LIN {X 0,Y 256.151,Z 298.388,A -85,B 0,C 180,E1 -18561.12,E2 -18561.12} C_VEL
LIN {X 0,Y 256.183,Z 298.389,A -85,B 0,C 180,E1 -18565.139,E2 -18565.139} C_VEL
LIN {X 0,Y 256.099,Z 298.396,A -85,B 0,C 180,E1 -18569.602,E2 -18569.602} C_VEL
LIN {X 0,Y 256.137,Z 298.525,A -85,B 0,C 180,E1 -18573.387,E2 -18573.387} C_VEL
LIN {X 0,Y 256.985,Z 302.055,A -85,B 0,C 180,E1 -18575.051,E2 -18575.051} C_VEL
LIN {X 0,Y 263.939,Z 316.937,A -85,B 0,C 180,E1 -18576.488,E2 -18576.488} C_VEL
LIN {X 0,Y 267.967,Z 326.974,A -85,B 0,C 180,E1 -18577.308,E2 -18577.308} C_VEL
LIN {X 0,Y 269.292,Z 334.674,A -85,B 0,C 180,E1 -18577.711,E2 -18577.711} C_VEL
LIN {X 0,Y 267.661,Z 378.993,A -85,B 0,C 180,E1 -18578.986,E2 -18578.986} C_VEL
LIN {X 0,Y 266.948,Z 389.558,A -85,B 0,C 180,E1 -18579.509,E2 -18579.509} C_VEL
LIN {X 0,Y 265.887,Z 401.083,A -85,B 0,C 180,E1 -18580.395,E2 -18580.395} C_VEL
LIN {X 0,Y 264.658,Z 410.377,A -85,B 0,C 180,E1 -18581.383,E2 -18581.383} C_VEL
LIN {X 0,Y 263.326,Z 418.675,A -85,B 0,C 180,E1 -18582.501,E2 -18582.501} C_VEL
LIN {X 0,Y 262.135,Z 425.481,A -85,B 0,C 180,E1 -18583.626,E2 -18583.626} C_VEL
LIN {X 0,Y 260.662,Z 432.609,A -85,B 0,C 180,E1 -18585.053,E2 -18585.053} C_VEL
LIN {X 0,Y 259.485,Z 437.896,A -85,B 0,C 180,E1 -18586.321,E2 -18586.321} C_VEL
LIN {X 0,Y 258.097,Z 444.114,A -85,B 0,C 180,E1 -18588.155,E2 -18588.155} C_VEL
LIN {X 0,Y 257.179,Z 448.17,A -85,B 0,C 180,E1 -18589.609,E2 -18589.609} C_VEL
LIN {X 0,Y 256.425,Z 451.313,A -85,B 0,C 180,E1 -18590.924,E2 -18590.924} C_VEL
LIN {X 0,Y 255.519,Z 455.024,A -85,B 0,C 180,E1 -18592.906,E2 -18592.906} C_VEL
LIN {X 0,Y 254.875,Z 457.473,A -85,B 0,C 180,E1 -18594.617,E2 -18594.617} C_VEL
LIN {X 0,Y 254.468,Z 459.361,A -85,B 0,C 180,E1 -18596.472,E2 -18596.472} C_VEL
LIN {X 0,Y 253.925,Z 460.797,A -85,B 0,C 180,E1 -18599.093,E2 -18599.093} C_VEL
LIN {X 0,Y 253.67,Z 460.823,A -85,B 0,C 180,E1 -18601.902,E2 -18601.902} C_VEL
LIN {X 0,Y 253.733,Z 460.029,A -85,B 0,C 180,E1 -18603.694,E2 -18603.694} C_VEL
LIN {X 0,Y 254.011,Z 458.128,A -85,B 0,C 180,E1 -18605.93,E2 -18605.93} C_VEL
LIN {X 0,Y 254.428,Z 455.249,A -85,B 0,C 180,E1 -18608.106,E2 -18608.106} C_VEL
LIN {X 0,Y 255.092,Z 450.342,A -85,B 0,C 180,E1 -18610.695,E2 -18610.695} C_VEL
LIN {X 0,Y 255.797,Z 444.962,A -85,B 0,C 180,E1 -18612.77,E2 -18612.77} C_VEL
LIN {X 0,Y 256.639,Z 439.307,A -85,B 0,C 180,E1 -18614.515,E2 -18614.515} C_VEL
LIN {X 0,Y 257.604,Z 432.621,A -85,B 0,C 180,E1 -18616.19,E2 -18616.19} C_VEL
LIN {X 0,Y 258.639,Z 425.015,A -85,B 0,C 180,E1 -18617.738,E2 -18617.738} C_VEL
LIN {X 0,Y 259.909,Z 415.481,A -85,B 0,C 180,E1 -18619.287,E2 -18619.287} C_VEL
LIN {X 0,Y 260.987,Z 405.524,A -85,B 0,C 180,E1 -18620.507,E2 -18620.507} C_VEL
LIN {X 0,Y 261.726,Z 395.897,A -85,B 0,C 180,E1 -18621.411,E2 -18621.411} C_VEL
LIN {X 0,Y 262.374,Z 386.398,A -85,B 0,C 180,E1 -18622.062,E2 -18622.062} C_VEL
LIN {X 0,Y 262.898,Z 376.662,A -85,B 0,C 180,E1 -18622.506,E2 -18622.506} C_VEL
LIN {X 0,Y 263.995,Z 331.197,A -85,B 0,C 180,E1 -18623.814,E2 -18623.814} C_VEL
LIN {X 0,Y 260.762,Z 313.544,A -85,B 0,C 180,E1 -18624.586,E2 -18624.586} C_VEL
LIN {X 0,Y 257.013,Z 301.84,A -85,B 0,C 180,E1 -18625.25,E2 -18625.25} C_VEL
LIN {X 0,Y 256.516,Z 298.349,A -85,B 0,C 180,E1 -18626.859,E2 -18626.859} C_VEL
LIN {X 0,Y 256.767,Z 298.316,A -85,B 0,C 180,E1 -18630,E2 -18630} C_VEL
LIN {X 0,Y 256.498,Z 298.345,A -85,B 0,C 180,E1 -18633.141,E2 -18633.141} C_VEL
LIN {X 0,Y 256.498,Z 298.346,A -85,B 0,C 180,E1 -18637.874,E2 -18637.874} C_VEL
LIN {X 0,Y 256.291,Z 298.369,A -85,B 0,C 180,E1 -18642.672,E2 -18642.672} C_VEL
LIN {X 0,Y 256.244,Z 298.379,A -85,B 0,C 180,E1 -18646.271,E2 -18646.271} C_VEL
LIN {X 0,Y 256.142,Z 298.377,A -85,B 0,C 180,E1 -18651.11,E2 -18651.11} C_VEL
LIN {X 0,Y 256.17,Z 298.388,A -85,B 0,C 180,E1 -18655.129,E2 -18655.129} C_VEL
LIN {X 0,Y 256.113,Z 298.394,A -85,B 0,C 180,E1 -18659.599,E2 -18659.599} C_VEL
LIN {X 0,Y 256.067,Z 298.399,A -85,B 0,C 180,E1 -18663.292,E2 -18663.292} C_VEL
LIN {X 0,Y 256.112,Z 298.398,A -85,B 0,C 180,E1 -18667.27,E2 -18667.27} C_VEL
LIN {X 0,Y 256.057,Z 298.4,A -85,B 0,C 180,E1 -18671.201,E2 -18671.201} C_VEL
LIN {X 0,Y 256.073,Z 298.399,A -85,B 0,C 180,E1 -18675.525,E2 -18675.525} C_VEL
LIN {X 0,Y 256.1,Z 298.394,A -85,B 0,C 180,E1 -18678.805,E2 -18678.805} C_VEL
LIN {X 0,Y 256.149,Z 298.383,A -85,B 0,C 180,E1 -18682.87,E2 -18682.87} C_VEL
LIN {X 0,Y 256.08,Z 298.391,A -85,B 0,C 180,E1 -18686.709,E2 -18686.709} C_VEL
LIN {X 0,Y 256.13,Z 298.39,A -85,B 0,C 180,E1 -18691.405,E2 -18691.405} C_VEL
LIN {X 0,Y 256.161,Z 298.384,A -85,B 0,C 180,E1 -18695.698,E2 -18695.698} C_VEL
LIN {X 0,Y 256.16,Z 298.374,A -85,B 0,C 180,E1 -18699.104,E2 -18699.104} C_VEL
LIN {X 0,Y 256.287,Z 298.369,A -85,B 0,C 180,E1 -18704.084,E2 -18704.084} C_VEL
LIN {X 0,Y 256.286,Z 298.371,A -85,B 0,C 180,E1 -18707.327,E2 -18707.327} C_VEL
LIN {X 0,Y 256.507,Z 298.339,A -85,B 0,C 180,E1 -18712.126,E2 -18712.126} C_VEL
LIN {X 0,Y 256.488,Z 298.34,A -85,B 0,C 180,E1 -18716.858,E2 -18716.858} C_VEL
LIN {X 0,Y 256.757,Z 298.31,A -85,B 0,C 180,E1 -18720,E2 -18720} C_VEL
LIN {X 0,Y 256.488,Z 298.35,A -85,B 0,C 180,E1 -18723.141,E2 -18723.141} C_VEL
LIN {X 0,Y 256.507,Z 298.337,A -85,B 0,C 180,E1 -18727.874,E2 -18727.874} C_VEL
LIN {X 0,Y 256.287,Z 298.368,A -85,B 0,C 180,E1 -18732.672,E2 -18732.672} C_VEL
LIN {X 0,Y 256.27,Z 298.375,A -85,B 0,C 180,E1 -18735.88,E2 -18735.88} C_VEL
LIN {X 0,Y 255.651,Z 298.459,A -85,B 0,C 180,E1 -18737.191,E2 -18737.191} C_VEL
LIN {X 0,Y 252.715,Z 298.819,A -85,B 0,C 180,E1 -18739.322,E2 -18739.322} C_VEL
LIN {X 0,Y 250.187,Z 299.124,A -85,B 0,C 180,E1 -18741.059,E2 -18741.059} C_VEL
LIN {X 0,Y 249.116,Z 299.262,A -85,B 0,C 180,E1 -18742.409,E2 -18742.409} C_VEL
LIN {X 0,Y 249.039,Z 299.268,A -85,B 0,C 180,E1 -18742.867,E2 -18742.867} C_VEL
LIN {X 0,Y 249.11,Z 299.265,A -85,B 0,C 180,E1 -18745.476,E2 -18745.476} C_VEL
LIN {X 0,Y 249.067,Z 299.268,A -85,B 0,C 180,E1 -18748.989,E2 -18748.989} C_VEL
LIN {X 0,Y 249.025,Z 299.279,A -85,B 0,C 180,E1 -18752.426,E2 -18752.426} C_VEL
LIN {X 0,Y 249.042,Z 299.277,A -85,B 0,C 180,E1 -18756.343,E2 -18756.343} C_VEL
LIN {X 0,Y 249.001,Z 299.27,A -85,B 0,C 180,E1 -18760.479,E2 -18760.479} C_VEL
LIN {X 0,Y 249.003,Z 299.282,A -85,B 0,C 180,E1 -18764.879,E2 -18764.879} C_VEL
LIN {X 0,Y 249.014,Z 299.277,A -85,B 0,C 180,E1 -18767.364,E2 -18767.364} C_VEL
LIN {X 0,Y 249.04,Z 299.274,A -85,B 0,C 180,E1 -18772.201,E2 -18772.201} C_VEL
LIN {X 0,Y 249.04,Z 299.274,A -85,B 0,C 180,E1 -18775.64,E2 -18775.64} C_VEL
LIN {X 0,Y 249.104,Z 299.285,A -85,B 0,C 180,E1 -18779.681,E2 -18779.681} C_VEL
LIN {X 0,Y 250.677,Z 307.76,A -85,B 0,C 180,E1 -18783.348,E2 -18783.348} C_VEL
LIN {X 0,Y 251.627,Z 313.3,A -85,B 0,C 180,E1 -18785.672,E2 -18785.672} C_VEL
LIN {X 0,Y 251.442,Z 315.01,A -85,B 0,C 180,E1 -18786.346,E2 -18786.346} C_VEL
LIN {X 0,Y 256.334,Z 351.638,A -85,B 0,C 180,E1 -18787.87,E2 -18787.87} C_VEL
LIN {X 0,Y 256.775,Z 358.082,A -85,B 0,C 180,E1 -18788.1,E2 -18788.1} C_VEL
LIN {X 0,Y 255.846,Z 392.247,A -85,B 0,C 180,E1 -18789.13,E2 -18789.13} C_VEL
LIN {X 0,Y 255.2,Z 402.545,A -85,B 0,C 180,E1 -18789.652,E2 -18789.652} C_VEL
LIN {X 0,Y 254.459,Z 410.782,A -85,B 0,C 180,E1 -18790.259,E2 -18790.259} C_VEL
LIN {X 0,Y 253.319,Z 422.12,A -85,B 0,C 180,E1 -18791.395,E2 -18791.395} C_VEL
LIN {X 0,Y 252.082,Z 432.063,A -85,B 0,C 180,E1 -18792.77,E2 -18792.77} C_VEL
LIN {X 0,Y 250.974,Z 440.032,A -85,B 0,C 180,E1 -18794.156,E2 -18794.156} C_VEL
LIN {X 0,Y 249.886,Z 447.476,A -85,B 0,C 180,E1 -18795.754,E2 -18795.754} C_VEL
LIN {X 0,Y 248.779,Z 455.022,A -85,B 0,C 180,E1 -18797.768,E2 -18797.768} C_VEL
LIN {X 0,Y 247.969,Z 460.929,A -85,B 0,C 180,E1 -18799.797,E2 -18799.797} C_VEL
LIN {X 0,Y 247.384,Z 465.565,A -85,B 0,C 180,E1 -18801.834,E2 -18801.834} C_VEL
LIN {X 0,Y 247.098,Z 468.571,A -85,B 0,C 180,E1 -18803.468,E2 -18803.468} C_VEL
LIN {X 0,Y 246.923,Z 470.901,A -85,B 0,C 180,E1 -18805.102,E2 -18805.102} C_VEL
LIN {X 0,Y 246.907,Z 472.628,A -85,B 0,C 180,E1 -18806.737,E2 -18806.737} C_VEL
LIN {X 0,Y 246.931,Z 473.843,A -85,B 0,C 180,E1 -18808.369,E2 -18808.369} C_VEL
LIN {X 0,Y 246.981,Z 474.572,A -85,B 0,C 180,E1 -18810,E2 -18810} C_VEL
LIN {X 0,Y 246.907,Z 474.817,A -85,B 0,C 180,E1 -18811.631,E2 -18811.631} C_VEL
LIN {X 0,Y 246.88,Z 474.471,A -85,B 0,C 180,E1 -18813.264,E2 -18813.264} C_VEL
LIN {X 0,Y 246.943,Z 473.512,A -85,B 0,C 180,E1 -18815.063,E2 -18815.063} C_VEL
LIN {X 0,Y 247.126,Z 472.282,A -85,B 0,C 180,E1 -18816.532,E2 -18816.532} C_VEL
LIN {X 0,Y 247.695,Z 469.279,A -85,B 0,C 180,E1 -18818.978,E2 -18818.978} C_VEL
LIN {X 0,Y 248.63,Z 465.018,A -85,B 0,C 180,E1 -18821.412,E2 -18821.412} C_VEL
LIN {X 0,Y 250.029,Z 459.189,A -85,B 0,C 180,E1 -18823.823,E2 -18823.823} C_VEL
LIN {X 0,Y 251.462,Z 452.925,A -85,B 0,C 180,E1 -18825.812,E2 -18825.812} C_VEL
LIN {X 0,Y 252.838,Z 446.82,A -85,B 0,C 180,E1 -18827.386,E2 -18827.386} C_VEL
LIN {X 0,Y 254.495,Z 439.407,A -85,B 0,C 180,E1 -18828.934,E2 -18828.934} C_VEL
LIN {X 0,Y 256.081,Z 431.486,A -85,B 0,C 180,E1 -18830.272,E2 -18830.272} C_VEL
LIN {X 0,Y 257.77,Z 421.644,A -85,B 0,C 180,E1 -18831.596,E2 -18831.596} C_VEL
LIN {X 0,Y 259.361,Z 410.129,A -85,B 0,C 180,E1 -18832.715,E2 -18832.715} C_VEL
LIN {X 0,Y 260.463,Z 400.369,A -85,B 0,C 180,E1 -18833.383,E2 -18833.383} C_VEL
LIN {X 0,Y 261.127,Z 391.422,A -85,B 0,C 180,E1 -18833.81,E2 -18833.81} C_VEL
LIN {X 0,Y 262.279,Z 357.245,A -85,B 0,C 180,E1 -18834.839,E2 -18834.839} C_VEL
LIN {X 0,Y 260.069,Z 341.118,A -85,B 0,C 180,E1 -18835.647,E2 -18835.647} C_VEL
LIN {X 0,Y 256.847,Z 324.506,A -85,B 0,C 180,E1 -18836.639,E2 -18836.639} C_VEL
LIN {X 0,Y 252.166,Z 313.492,A -85,B 0,C 180,E1 -18837.724,E2 -18837.724} C_VEL
LIN {X 0,Y 250.557,Z 305.695,A -85,B 0,C 180,E1 -18841.258,E2 -18841.258} C_VEL
LIN {X 0,Y 249.055,Z 299.276,A -85,B 0,C 180,E1 -18844.357,E2 -18844.357} C_VEL
LIN {X 0,Y 249.022,Z 299.285,A -85,B 0,C 180,E1 -18848.38,E2 -18848.38} C_VEL
LIN {X 0,Y 248.997,Z 299.285,A -85,B 0,C 180,E1 -18852.79,E2 -18852.79} C_VEL
LIN {X 0,Y 249.004,Z 299.283,A -85,B 0,C 180,E1 -18857.361,E2 -18857.361} C_VEL
LIN {X 0,Y 249.022,Z 299.274,A -85,B 0,C 180,E1 -18861.619,E2 -18861.619} C_VEL
LIN {X 0,Y 249.039,Z 299.275,A -85,B 0,C 180,E1 -18865.639,E2 -18865.639} C_VEL
LIN {X 0,Y 249.046,Z 299.273,A -85,B 0,C 180,E1 -18869.473,E2 -18869.473} C_VEL
LIN {X 0,Y 249.063,Z 299.258,A -85,B 0,C 180,E1 -18873.161,E2 -18873.161} C_VEL
LIN {X 0,Y 249.054,Z 299.267,A -85,B 0,C 180,E1 -18876.73,E2 -18876.73} C_VEL
LIN {X 0,Y 249.102,Z 299.263,A -85,B 0,C 180,E1 -18880.211,E2 -18880.211} C_VEL
LIN {X 0,Y 249.236,Z 299.237,A -85,B 0,C 180,E1 -18883.622,E2 -18883.622} C_VEL
LIN {X 0,Y 249.236,Z 299.246,A -85,B 0,C 180,E1 -18888.616,E2 -18888.616} C_VEL
LIN {X 0,Y 249.447,Z 299.214,A -85,B 0,C 180,E1 -18891.902,E2 -18891.902} C_VEL
LIN {X 0,Y 249.284,Z 299.235,A -85,B 0,C 180,E1 -18895.148,E2 -18895.148} C_VEL
LIN {X 0,Y 249.666,Z 299.189,A -85,B 0,C 180,E1 -18898.387,E2 -18898.387} C_VEL
LIN {X 0,Y 249.666,Z 299.183,A -85,B 0,C 180,E1 -18901.613,E2 -18901.613} C_VEL
LIN {X 0,Y 249.418,Z 299.222,A -85,B 0,C 180,E1 -18906.537,E2 -18906.537} C_VEL
LIN {X 0,Y 249.337,Z 299.24,A -85,B 0,C 180,E1 -18909.737,E2 -18909.737} C_VEL
LIN {X 0,Y 249.19,Z 299.258,A -85,B 0,C 180,E1 -18914.704,E2 -18914.704} C_VEL
LIN {X 0,Y 249.129,Z 299.266,A -85,B 0,C 180,E1 -18918.078,E2 -18918.078} C_VEL
LIN {X 0,Y 249.081,Z 299.271,A -85,B 0,C 180,E1 -18921.519,E2 -18921.519} C_VEL
LIN {X 0,Y 249.125,Z 299.27,A -85,B 0,C 180,E1 -18925.483,E2 -18925.483} C_VEL
LIN {X 0,Y 249.068,Z 299.27,A -85,B 0,C 180,E1 -18928.99,E2 -18928.99} C_VEL
LIN {X 0,Y 249.047,Z 299.309,A -85,B 0,C 180,E1 -18932.543,E2 -18932.543} C_VEL
LIN {X 0,Y 249.893,Z 302.544,A -85,B 0,C 180,E1 -18934.045,E2 -18934.045} C_VEL
LIN {X 0,Y 257.145,Z 317.447,A -85,B 0,C 180,E1 -18935.608,E2 -18935.608} C_VEL
LIN {X 0,Y 262.017,Z 329.387,A -85,B 0,C 180,E1 -18936.659,E2 -18936.659} C_VEL
LIN {X 0,Y 263.065,Z 335.339,A -85,B 0,C 180,E1 -18936.986,E2 -18936.986} C_VEL
LIN {X 0,Y 261.363,Z 379.31,A -85,B 0,C 180,E1 -18938.279,E2 -18938.279} C_VEL
LIN {X 0,Y 260.618,Z 390.029,A -85,B 0,C 180,E1 -18938.825,E2 -18938.825} C_VEL
LIN {X 0,Y 259.451,Z 401.845,A -85,B 0,C 180,E1 -18939.772,E2 -18939.772} C_VEL
LIN {X 0,Y 258.13,Z 411.2,A -85,B 0,C 180,E1 -18940.802,E2 -18940.802} C_VEL
LIN {X 0,Y 256.907,Z 418.493,A -85,B 0,C 180,E1 -18941.804,E2 -18941.804} C_VEL
LIN {X 0,Y 255.623,Z 425.55,A -85,B 0,C 180,E1 -18942.99,E2 -18942.99} C_VEL
LIN {X 0,Y 253.948,Z 433.158,A -85,B 0,C 180,E1 -18944.553,E2 -18944.553} C_VEL
LIN {X 0,Y 252.641,Z 438.698,A -85,B 0,C 180,E1 -18945.938,E2 -18945.938} C_VEL
LIN {X 0,Y 251.531,Z 443.472,A -85,B 0,C 180,E1 -18947.364,E2 -18947.364} C_VEL
LIN {X 0,Y 250.222,Z 448.785,A -85,B 0,C 180,E1 -18949.319,E2 -18949.319} C_VEL
LIN {X 0,Y 249.459,Z 451.837,A -85,B 0,C 180,E1 -18950.664,E2 -18950.664} C_VEL
LIN {X 0,Y 248.684,Z 454.871,A -85,B 0,C 180,E1 -18952.308,E2 -18952.308} C_VEL
LIN {X 0,Y 247.837,Z 457.857,A -85,B 0,C 180,E1 -18954.458,E2 -18954.458} C_VEL
LIN {X 0,Y 247.155,Z 460.258,A -85,B 0,C 180,E1 -18957.299,E2 -18957.299} C_VEL
LIN {X 0,Y 246.815,Z 461.045,A -85,B 0,C 180,E1 -18959.168,E2 -18959.168} C_VEL
LIN {X 0,Y 246.584,Z 460.961,A -85,B 0,C 180,E1 -18962.074,E2 -18962.074} C_VEL
LIN {X 0,Y 246.72,Z 459.547,A -85,B 0,C 180,E1 -18964.705,E2 -18964.705} C_VEL
LIN {X 0,Y 247.034,Z 457.72,A -85,B 0,C 180,E1 -18966.529,E2 -18966.529} C_VEL
LIN {X 0,Y 247.508,Z 454.157,A -85,B 0,C 180,E1 -18968.98,E2 -18968.98} C_VEL
LIN {X 0,Y 248.217,Z 449.125,A -85,B 0,C 180,E1 -18971.426,E2 -18971.426} C_VEL
LIN {X 0,Y 248.849,Z 444.55,A -85,B 0,C 180,E1 -18973.174,E2 -18973.174} C_VEL
LIN {X 0,Y 249.717,Z 438.959,A -85,B 0,C 180,E1 -18974.911,E2 -18974.911} C_VEL
LIN {X 0,Y 250.45,Z 434.013,A -85,B 0,C 180,E1 -18976.201,E2 -18976.201} C_VEL
LIN {X 0,Y 251.365,Z 427.852,A -85,B 0,C 180,E1 -18977.558,E2 -18977.558} C_VEL
LIN {X 0,Y 252.429,Z 420.063,A -85,B 0,C 180,E1 -18978.965,E2 -18978.965} C_VEL
LIN {X 0,Y 253.514,Z 411.395,A -85,B 0,C 180,E1 -18980.224,E2 -18980.224} C_VEL
LIN {X 0,Y 254.447,Z 402.338,A -85,B 0,C 180,E1 -18981.262,E2 -18981.262} C_VEL
LIN {X 0,Y 255.343,Z 390.86,A -85,B 0,C 180,E1 -18982.247,E2 -18982.247} C_VEL
LIN {X 0,Y 255.961,Z 380.029,A -85,B 0,C 180,E1 -18982.84,E2 -18982.84} C_VEL
LIN {X 0,Y 256.723,Z 354.048,A -85,B 0,C 180,E1 -18983.645,E2 -18983.645} C_VEL
LIN {X 0,Y 257.202,Z 331.869,A -85,B 0,C 180,E1 -18984.292,E2 -18984.292} C_VEL
LIN {X 0,Y 254.222,Z 315.471,A -85,B 0,C 180,E1 -18985.033,E2 -18985.033} C_VEL
LIN {X 0,Y 249.85,Z 301.947,A -85,B 0,C 180,E1 -18985.867,E2 -18985.867} C_VEL
LIN {X 0,Y 249.495,Z 299.225,A -85,B 0,C 180,E1 -18987.175,E2 -18987.175} C_VEL
LIN {X 0,Y 249.73,Z 299.193,A -85,B 0,C 180,E1 -18990,E2 -18990} C_VEL
LIN {X 0,Y 249.434,Z 299.225,A -85,B 0,C 180,E1 -18993.23,E2 -18993.23} C_VEL
LIN {X 0,Y 249.439,Z 299.225,A -85,B 0,C 180,E1 -18996.471,E2 -18996.471} C_VEL
LIN {X 0,Y 249.345,Z 299.238,A -85,B 0,C 180,E1 -18999.736,E2 -18999.736} C_VEL
LIN {X 0,Y 249.184,Z 299.258,A -85,B 0,C 180,E1 -19004.704,E2 -19004.704} C_VEL
LIN {X 0,Y 249.113,Z 299.265,A -85,B 0,C 180,E1 -19008.079,E2 -19008.079} C_VEL
LIN {X 0,Y 249.081,Z 299.254,A -85,B 0,C 180,E1 -19011.518,E2 -19011.518} C_VEL
LIN {X 0,Y 249.117,Z 299.265,A -85,B 0,C 180,E1 -19015.475,E2 -19015.475} C_VEL
LIN {X 0,Y 249.083,Z 299.274,A -85,B 0,C 180,E1 -19018.992,E2 -19018.992} C_VEL
LIN {X 0,Y 249.03,Z 299.273,A -85,B 0,C 180,E1 -19022.425,E2 -19022.425} C_VEL
LIN {X 0,Y 249.028,Z 299.276,A -85,B 0,C 180,E1 -19026.345,E2 -19026.345} C_VEL
LIN {X 0,Y 249.005,Z 299.276,A -85,B 0,C 180,E1 -19030.477,E2 -19030.477} C_VEL
LIN {X 0,Y 249.016,Z 299.274,A -85,B 0,C 180,E1 -19034.874,E2 -19034.874} C_VEL
LIN {X 0,Y 249.059,Z 299.273,A -85,B 0,C 180,E1 -19037.372,E2 -19037.372} C_VEL
LIN {X 0,Y 249.048,Z 299.273,A -85,B 0,C 180,E1 -19041.623,E2 -19041.623} C_VEL
LIN {X 0,Y 249.057,Z 299.263,A -85,B 0,C 180,E1 -19045.641,E2 -19045.641} C_VEL
LIN {X 0,Y 249.046,Z 299.272,A -85,B 0,C 180,E1 -19049.472,E2 -19049.472} C_VEL
LIN {X 0,Y 249.068,Z 299.269,A -85,B 0,C 180,E1 -19053.161,E2 -19053.161} C_VEL
LIN {X 0,Y 249.073,Z 299.263,A -85,B 0,C 180,E1 -19056.732,E2 -19056.732} C_VEL
LIN {X 0,Y 249.104,Z 299.255,A -85,B 0,C 180,E1 -19060.211,E2 -19060.211} C_VEL
LIN {X 0,Y 249.236,Z 299.246,A -85,B 0,C 180,E1 -19063.621,E2 -19063.621} C_VEL
LIN {X 0,Y 249.237,Z 299.253,A -85,B 0,C 180,E1 -19068.616,E2 -19068.616} C_VEL
LIN {X 0,Y 249.447,Z 299.218,A -85,B 0,C 180,E1 -19071.902,E2 -19071.902} C_VEL
LIN {X 0,Y 249.286,Z 299.234,A -85,B 0,C 180,E1 -19075.148,E2 -19075.148} C_VEL
LIN {X 0,Y 249.667,Z 299.191,A -85,B 0,C 180,E1 -19078.387,E2 -19078.387} C_VEL
LIN {X 0,Y 249.667,Z 299.196,A -85,B 0,C 180,E1 -19081.613,E2 -19081.613} C_VEL
LIN {X 0,Y 249.445,Z 299.219,A -85,B 0,C 180,E1 -19086.471,E2 -19086.471} C_VEL
LIN {X 0,Y 249.337,Z 299.231,A -85,B 0,C 180,E1 -19089.737,E2 -19089.737} C_VEL
LIN {X 0,Y 249.19,Z 299.254,A -85,B 0,C 180,E1 -19094.704,E2 -19094.704} C_VEL
LIN {X 0,Y 249.127,Z 299.262,A -85,B 0,C 180,E1 -19098.078,E2 -19098.078} C_VEL
LIN {X 0,Y 249.078,Z 299.264,A -85,B 0,C 180,E1 -19101.519,E2 -19101.519} C_VEL
LIN {X 0,Y 249.039,Z 299.268,A -85,B 0,C 180,E1 -19102.867,E2 -19102.867} C_VEL
LIN {X 0,Y 248.407,Z 299.355,A -85,B 0,C 180,E1 -19104.218,E2 -19104.218} C_VEL
LIN {X 0,Y 245.585,Z 299.71,A -85,B 0,C 180,E1 -19106.419,E2 -19106.419} C_VEL
LIN {X 0,Y 243.149,Z 300.01,A -85,B 0,C 180,E1 -19108.212,E2 -19108.212} C_VEL
LIN {X 0,Y 242.071,Z 300.14,A -85,B 0,C 180,E1 -19109.602,E2 -19109.602} C_VEL
LIN {X 0,Y 241.966,Z 300.15,A -85,B 0,C 180,E1 -19110.074,E2 -19110.074} C_VEL
LIN {X 0,Y 241.975,Z 300.154,A -85,B 0,C 180,E1 -19113.493,E2 -19113.493} C_VEL
LIN {X 0,Y 241.984,Z 300.151,A -85,B 0,C 180,E1 -19117.583,E2 -19117.583} C_VEL
LIN {X 0,Y 241.934,Z 300.149,A -85,B 0,C 180,E1 -19121.923,E2 -19121.923} C_VEL
LIN {X 0,Y 241.933,Z 300.162,A -85,B 0,C 180,E1 -19126.571,E2 -19126.571} C_VEL
LIN {X 0,Y 241.953,Z 300.157,A -85,B 0,C 180,E1 -19130.282,E2 -19130.282} C_VEL
LIN {X 0,Y 241.978,Z 300.155,A -85,B 0,C 180,E1 -19134.489,E2 -19134.489} C_VEL
LIN {X 0,Y 242.05,Z 300.187,A -85,B 0,C 180,E1 -19139.343,E2 -19139.343} C_VEL
LIN {X 0,Y 243.612,Z 308.448,A -85,B 0,C 180,E1 -19143.033,E2 -19143.033} C_VEL
LIN {X 0,Y 244.59,Z 314.808,A -85,B 0,C 180,E1 -19145.765,E2 -19145.765} C_VEL
LIN {X 0,Y 249.536,Z 351.779,A -85,B 0,C 180,E1 -19147.364,E2 -19147.364} C_VEL
LIN {X 0,Y 250.027,Z 358.648,A -85,B 0,C 180,E1 -19147.62,E2 -19147.62} C_VEL
LIN {X 0,Y 249.05,Z 392.711,A -85,B 0,C 180,E1 -19148.681,E2 -19148.681} C_VEL
LIN {X 0,Y 248.338,Z 402.93,A -85,B 0,C 180,E1 -19149.222,E2 -19149.222} C_VEL
LIN {X 0,Y 247.56,Z 411.883,A -85,B 0,C 180,E1 -19149.92,E2 -19149.92} C_VEL
LIN {X 0,Y 246.383,Z 422.609,A -85,B 0,C 180,E1 -19151.067,E2 -19151.067} C_VEL
LIN {X 0,Y 245.253,Z 431.184,A -85,B 0,C 180,E1 -19152.274,E2 -19152.274} C_VEL
LIN {X 0,Y 244.147,Z 439.274,A -85,B 0,C 180,E1 -19153.701,E2 -19153.701} C_VEL
LIN {X 0,Y 243.235,Z 445.088,A -85,B 0,C 180,E1 -19154.928,E2 -19154.928} C_VEL
LIN {X 0,Y 242.25,Z 451.571,A -85,B 0,C 180,E1 -19156.58,E2 -19156.58} C_VEL
LIN {X 0,Y 241.427,Z 456.953,A -85,B 0,C 180,E1 -19158.243,E2 -19158.243} C_VEL
LIN {X 0,Y 240.815,Z 461.437,A -85,B 0,C 180,E1 -19159.915,E2 -19159.915} C_VEL
LIN {X 0,Y 240.18,Z 466.695,A -85,B 0,C 180,E1 -19162.434,E2 -19162.434} C_VEL
LIN {X 0,Y 239.917,Z 469.386,A -85,B 0,C 180,E1 -19164.115,E2 -19164.115} C_VEL
LIN {X 0,Y 239.811,Z 472.321,A -85,B 0,C 180,E1 -19166.64,E2 -19166.64} C_VEL
LIN {X 0,Y 239.842,Z 473.581,A -85,B 0,C 180,E1 -19168.321,E2 -19168.321} C_VEL
LIN {X 0,Y 239.911,Z 474.354,A -85,B 0,C 180,E1 -19170,E2 -19170} C_VEL
LIN {X 0,Y 239.819,Z 474.622,A -85,B 0,C 180,E1 -19171.679,E2 -19171.679} C_VEL
LIN {X 0,Y 239.786,Z 474.295,A -85,B 0,C 180,E1 -19173.36,E2 -19173.36} C_VEL
LIN {X 0,Y 239.843,Z 473.482,A -85,B 0,C 180,E1 -19175.043,E2 -19175.043} C_VEL
LIN {X 0,Y 240.063,Z 472.199,A -85,B 0,C 180,E1 -19176.725,E2 -19176.725} C_VEL
LIN {X 0,Y 240.684,Z 469.252,A -85,B 0,C 180,E1 -19179.241,E2 -19179.241} C_VEL
LIN {X 0,Y 241.312,Z 466.584,A -85,B 0,C 180,E1 -19180.912,E2 -19180.912} C_VEL
LIN {X 0,Y 242.59,Z 461.376,A -85,B 0,C 180,E1 -19183.401,E2 -19183.401} C_VEL
LIN {X 0,Y 244.366,Z 454.556,A -85,B 0,C 180,E1 -19185.856,E2 -19185.856} C_VEL
LIN {X 0,Y 246.092,Z 447.123,A -85,B 0,C 180,E1 -19187.878,E2 -19187.878} C_VEL
LIN {X 0,Y 247.808,Z 439.809,A -85,B 0,C 180,E1 -19189.465,E2 -19189.465} C_VEL
LIN {X 0,Y 249.452,Z 432.008,A -85,B 0,C 180,E1 -19190.835,E2 -19190.835} C_VEL
LIN {X 0,Y 250.771,Z 425.297,A -85,B 0,C 180,E1 -19191.797,E2 -19191.797} C_VEL
LIN {X 0,Y 252.017,Z 417.159,A -85,B 0,C 180,E1 -19192.763,E2 -19192.763} C_VEL
LIN {X 0,Y 253.27,Z 408.235,A -85,B 0,C 180,E1 -19193.574,E2 -19193.574} C_VEL
LIN {X 0,Y 254.377,Z 398.369,A -85,B 0,C 180,E1 -19194.227,E2 -19194.227} C_VEL
LIN {X 0,Y 255.136,Z 387.374,A -85,B 0,C 180,E1 -19194.706,E2 -19194.706} C_VEL
LIN {X 0,Y 256.07,Z 358.134,A -85,B 0,C 180,E1 -19195.587,E2 -19195.587} C_VEL
LIN {X 0,Y 253.976,Z 342.579,A -85,B 0,C 180,E1 -19196.402,E2 -19196.402} C_VEL
LIN {X 0,Y 250.998,Z 327.162,A -85,B 0,C 180,E1 -19197.361,E2 -19197.361} C_VEL
LIN {X 0,Y 245.986,Z 315.969,A -85,B 0,C 180,E1 -19198.511,E2 -19198.511} C_VEL
LIN {X 0,Y 244.934,Z 313.227,A -85,B 0,C 180,E1 -19198.826,E2 -19198.826} C_VEL
LIN {X 0,Y 243.451,Z 306.289,A -85,B 0,C 180,E1 -19202.123,E2 -19202.123} C_VEL
LIN {X 0,Y 242,Z 300.153,A -85,B 0,C 180,E1 -19205.252,E2 -19205.252} C_VEL
LIN {X 0,Y 241.953,Z 300.163,A -85,B 0,C 180,E1 -19209.718,E2 -19209.718} C_VEL
LIN {X 0,Y 241.914,Z 300.169,A -85,B 0,C 180,E1 -19214.204,E2 -19214.204} C_VEL
LIN {X 0,Y 241.929,Z 300.159,A -85,B 0,C 180,E1 -19218.076,E2 -19218.076} C_VEL
LIN {X 0,Y 241.987,Z 300.145,A -85,B 0,C 180,E1 -19222.418,E2 -19222.418} C_VEL
LIN {X 0,Y 241.976,Z 300.148,A -85,B 0,C 180,E1 -19226.507,E2 -19226.507} C_VEL
LIN {X 0,Y 242.031,Z 300.146,A -85,B 0,C 180,E1 -19230.587,E2 -19230.587} C_VEL
LIN {X 0,Y 242.062,Z 300.138,A -85,B 0,C 180,E1 -19234.183,E2 -19234.183} C_VEL
LIN {X 0,Y 242.019,Z 300.134,A -85,B 0,C 180,E1 -19238.313,E2 -19238.313} C_VEL
LIN {X 0,Y 242.157,Z 300.122,A -85,B 0,C 180,E1 -19243.278,E2 -19243.278} C_VEL
LIN {X 0,Y 242.173,Z 300.129,A -85,B 0,C 180,E1 -19248.279,E2 -19248.279} C_VEL
LIN {X 0,Y 242.393,Z 300.089,A -85,B 0,C 180,E1 -19251.665,E2 -19251.665} C_VEL
LIN {X 0,Y 242.245,Z 300.113,A -85,B 0,C 180,E1 -19255.007,E2 -19255.007} C_VEL
LIN {X 0,Y 242.627,Z 300.066,A -85,B 0,C 180,E1 -19258.34,E2 -19258.34} C_VEL
LIN {X 0,Y 242.626,Z 300.06,A -85,B 0,C 180,E1 -19261.66,E2 -19261.66} C_VEL
LIN {X 0,Y 242.393,Z 300.095,A -85,B 0,C 180,E1 -19266.66,E2 -19266.66} C_VEL
LIN {X 0,Y 242.261,Z 300.12,A -85,B 0,C 180,E1 -19270.024,E2 -19270.024} C_VEL
LIN {X 0,Y 242.149,Z 300.136,A -85,B 0,C 180,E1 -19275.142,E2 -19275.142} C_VEL
LIN {X 0,Y 242.064,Z 300.148,A -85,B 0,C 180,E1 -19278.625,E2 -19278.625} C_VEL
LIN {X 0,Y 242.007,Z 300.158,A -85,B 0,C 180,E1 -19282.181,E2 -19282.181} C_VEL
LIN {X 0,Y 242.062,Z 300.146,A -85,B 0,C 180,E1 -19285.839,E2 -19285.839} C_VEL
LIN {X 0,Y 242.002,Z 300.152,A -85,B 0,C 180,E1 -19289.584,E2 -19289.584} C_VEL
LIN {X 0,Y 242.021,Z 300.363,A -85,B 0,C 180,E1 -19291.754,E2 -19291.754} C_VEL
LIN {X 0,Y 242.588,Z 302.562,A -85,B 0,C 180,E1 -19292.894,E2 -19292.894} C_VEL
LIN {X 0,Y 250.724,Z 318.867,A -85,B 0,C 180,E1 -19294.755,E2 -19294.755} C_VEL
LIN {X 0,Y 256.206,Z 332.32,A -85,B 0,C 180,E1 -19295.994,E2 -19295.994} C_VEL
LIN {X 0,Y 256.898,Z 337.05,A -85,B 0,C 180,E1 -19296.249,E2 -19296.249} C_VEL
LIN {X 0,Y 255.208,Z 378.649,A -85,B 0,C 180,E1 -19297.497,E2 -19297.497} C_VEL
LIN {X 0,Y 254.577,Z 387.962,A -85,B 0,C 180,E1 -19297.956,E2 -19297.956} C_VEL
LIN {X 0,Y 253.803,Z 396.138,A -85,B 0,C 180,E1 -19298.534,E2 -19298.534} C_VEL
LIN {X 0,Y 252.649,Z 405.354,A -85,B 0,C 180,E1 -19299.399,E2 -19299.399} C_VEL
LIN {X 0,Y 251.201,Z 414.434,A -85,B 0,C 180,E1 -19300.502,E2 -19300.502} C_VEL
LIN {X 0,Y 249.198,Z 425.241,A -85,B 0,C 180,E1 -19302.244,E2 -19302.244} C_VEL
LIN {X 0,Y 247.409,Z 433.091,A -85,B 0,C 180,E1 -19303.88,E2 -19303.88} C_VEL
LIN {X 0,Y 245.716,Z 439.893,A -85,B 0,C 180,E1 -19305.648,E2 -19305.648} C_VEL
LIN {X 0,Y 244.306,Z 445.511,A -85,B 0,C 180,E1 -19307.467,E2 -19307.467} C_VEL
LIN {X 0,Y 242.97,Z 450.518,A -85,B 0,C 180,E1 -19309.493,E2 -19309.493} C_VEL
LIN {X 0,Y 241.541,Z 455.708,A -85,B 0,C 180,E1 -19312.338,E2 -19312.338} C_VEL
LIN {X 0,Y 240.649,Z 458.772,A -85,B 0,C 180,E1 -19314.858,E2 -19314.858} C_VEL
LIN {X 0,Y 240.285,Z 460.013,A -85,B 0,C 180,E1 -19316.241,E2 -19316.241} C_VEL
LIN {X 0,Y 239.879,Z 461.076,A -85,B 0,C 180,E1 -19318.173,E2 -19318.173} C_VEL
LIN {X 0,Y 239.601,Z 461.444,A -85,B 0,C 180,E1 -19320.091,E2 -19320.091} C_VEL
LIN {X 0,Y 239.498,Z 461.152,A -85,B 0,C 180,E1 -19321.998,E2 -19321.998} C_VEL
LIN {X 0,Y 239.558,Z 460.231,A -85,B 0,C 180,E1 -19323.893,E2 -19323.893} C_VEL
LIN {X 0,Y 239.968,Z 457.736,A -85,B 0,C 180,E1 -19326.711,E2 -19326.711} C_VEL
LIN {X 0,Y 240.467,Z 453.989,A -85,B 0,C 180,E1 -19329.269,E2 -19329.269} C_VEL
LIN {X 0,Y 241.205,Z 448.953,A -85,B 0,C 180,E1 -19331.747,E2 -19331.747} C_VEL
LIN {X 0,Y 241.873,Z 444.391,A -85,B 0,C 180,E1 -19333.51,E2 -19333.51} C_VEL
LIN {X 0,Y 242.795,Z 438.612,A -85,B 0,C 180,E1 -19335.329,E2 -19335.329} C_VEL
LIN {X 0,Y 244.048,Z 430.632,A -85,B 0,C 180,E1 -19337.351,E2 -19337.351} C_VEL
LIN {X 0,Y 245.299,Z 421.966,A -85,B 0,C 180,E1 -19339.059,E2 -19339.059} C_VEL
LIN {X 0,Y 246.391,Z 413.673,A -85,B 0,C 180,E1 -19340.353,E2 -19340.353} C_VEL
LIN {X 0,Y 247.368,Z 405.095,A -85,B 0,C 180,E1 -19341.422,E2 -19341.422} C_VEL
LIN {X 0,Y 248.103,Z 396.314,A -85,B 0,C 180,E1 -19342.282,E2 -19342.282} C_VEL
LIN {X 0,Y 248.792,Z 387.04,A -85,B 0,C 180,E1 -19342.954,E2 -19342.954} C_VEL
LIN {X 0,Y 249.327,Z 377.562,A -85,B 0,C 180,E1 -19343.418,E2 -19343.418} C_VEL
LIN {X 0,Y 250.44,Z 332.622,A -85,B 0,C 180,E1 -19344.791,E2 -19344.791} C_VEL
LIN {X 0,Y 247.608,Z 317.073,A -85,B 0,C 180,E1 -19345.514,E2 -19345.514} C_VEL
LIN {X 0,Y 242.749,Z 302.186,A -85,B 0,C 180,E1 -19346.447,E2 -19346.447} C_VEL
LIN {X 0,Y 242.521,Z 300.094,A -85,B 0,C 180,E1 -19347.509,E2 -19347.509} C_VEL
LIN {X 0,Y 242.694,Z 300.069,A -85,B 0,C 180,E1 -19350,E2 -19350} C_VEL
LIN {X 0,Y 242.637,Z 300.076,A -85,B 0,C 180,E1 -19351.66,E2 -19351.66} C_VEL
LIN {X 0,Y 242.411,Z 300.1,A -85,B 0,C 180,E1 -19356.659,E2 -19356.659} C_VEL
LIN {X 0,Y 242.269,Z 300.121,A -85,B 0,C 180,E1 -19360.023,E2 -19360.023} C_VEL
LIN {X 0,Y 242.14,Z 300.133,A -85,B 0,C 180,E1 -19365.142,E2 -19365.142} C_VEL
LIN {X 0,Y 242.05,Z 300.143,A -85,B 0,C 180,E1 -19368.625,E2 -19368.625} C_VEL
LIN {X 0,Y 242.005,Z 300.136,A -85,B 0,C 180,E1 -19372.18,E2 -19372.18} C_VEL
LIN {X 0,Y 242.067,Z 300.142,A -85,B 0,C 180,E1 -19375.837,E2 -19375.837} C_VEL
LIN {X 0,Y 242.03,Z 300.149,A -85,B 0,C 180,E1 -19379.579,E2 -19379.579} C_VEL
LIN {X 0,Y 241.979,Z 300.153,A -85,B 0,C 180,E1 -19383.492,E2 -19383.492} C_VEL
LIN {X 0,Y 241.985,Z 300.155,A -85,B 0,C 180,E1 -19387.581,E2 -19387.581} C_VEL
LIN {X 0,Y 241.941,Z 300.151,A -85,B 0,C 180,E1 -19391.92,E2 -19391.92} C_VEL
LIN {X 0,Y 241.988,Z 300.151,A -85,B 0,C 180,E1 -19396.556,E2 -19396.556} C_VEL
LIN {X 0,Y 242.004,Z 300.149,A -85,B 0,C 180,E1 -19400.29,E2 -19400.29} C_VEL
LIN {X 0,Y 242.033,Z 300.135,A -85,B 0,C 180,E1 -19404.497,E2 -19404.497} C_VEL
LIN {X 0,Y 241.971,Z 300.153,A -85,B 0,C 180,E1 -19408.479,E2 -19408.479} C_VEL
LIN {X 0,Y 242.002,Z 300.153,A -85,B 0,C 180,E1 -19412.312,E2 -19412.312} C_VEL
LIN {X 0,Y 242.052,Z 300.143,A -85,B 0,C 180,E1 -19416.015,E2 -19416.015} C_VEL
LIN {X 0,Y 242.031,Z 300.132,A -85,B 0,C 180,E1 -19419.607,E2 -19419.607} C_VEL
LIN {X 0,Y 242.158,Z 300.128,A -85,B 0,C 180,E1 -19423.278,E2 -19423.278} C_VEL
LIN {X 0,Y 242.173,Z 300.13,A -85,B 0,C 180,E1 -19428.279,E2 -19428.279} C_VEL
LIN {X 0,Y 242.393,Z 300.096,A -85,B 0,C 180,E1 -19431.664,E2 -19431.664} C_VEL
LIN {X 0,Y 242.247,Z 300.109,A -85,B 0,C 180,E1 -19435.007,E2 -19435.007} C_VEL
LIN {X 0,Y 242.628,Z 300.067,A -85,B 0,C 180,E1 -19438.34,E2 -19438.34} C_VEL
LIN {X 0,Y 242.628,Z 300.073,A -85,B 0,C 180,E1 -19441.66,E2 -19441.66} C_VEL
LIN {X 0,Y 242.415,Z 300.095,A -85,B 0,C 180,E1 -19446.659,E2 -19446.659} C_VEL
LIN {X 0,Y 242.261,Z 300.111,A -85,B 0,C 180,E1 -19450.024,E2 -19450.024} C_VEL
LIN {X 0,Y 242.15,Z 300.133,A -85,B 0,C 180,E1 -19455.142,E2 -19455.142} C_VEL
LIN {X 0,Y 242.062,Z 300.14,A -85,B 0,C 180,E1 -19458.625,E2 -19458.625} C_VEL
LIN {X 0,Y 241.985,Z 300.148,A -85,B 0,C 180,E1 -19462.869,E2 -19462.869} C_VEL
LIN {X 0,Y 242.061,Z 300.146,A -85,B 0,C 180,E1 -19465.839,E2 -19465.839} C_VEL
LIN {X 0,Y 241.966,Z 300.15,A -85,B 0,C 180,E1 -19470.074,E2 -19470.074} C_VEL
LIN {X 0,Y 241.26,Z 300.241,A -85,B 0,C 180,E1 -19471.463,E2 -19471.463} C_VEL
LIN {X 0,Y 238.414,Z 300.599,A -85,B 0,C 180,E1 -19473.731,E2 -19473.731} C_VEL
LIN {X 0,Y 236.014,Z 300.897,A -85,B 0,C 180,E1 -19475.578,E2 -19475.578} C_VEL
LIN {X 0,Y 234.973,Z 301.024,A -85,B 0,C 180,E1 -19477.01,E2 -19477.01} C_VEL
LIN {X 0,Y 234.881,Z 301.03,A -85,B 0,C 180,E1 -19477.496,E2 -19477.496} C_VEL
LIN {X 0,Y 234.879,Z 301.026,A -85,B 0,C 180,E1 -19481.581,E2 -19481.581} C_VEL
LIN {X 0,Y 234.894,Z 301.036,A -85,B 0,C 180,E1 -19485.896,E2 -19485.896} C_VEL
LIN {X 0,Y 234.881,Z 301.042,A -85,B 0,C 180,E1 -19488.833,E2 -19488.833} C_VEL
LIN {X 0,Y 234.915,Z 301.037,A -85,B 0,C 180,E1 -19491.079,E2 -19491.079} C_VEL
LIN {X 0,Y 234.923,Z 301.034,A -85,B 0,C 180,E1 -19495.362,E2 -19495.362} C_VEL
LIN {X 0,Y 235.014,Z 301.135,A -85,B 0,C 180,E1 -19499.009,E2 -19499.009} C_VEL
LIN {X 0,Y 236.638,Z 309.781,A -85,B 0,C 180,E1 -19502.996,E2 -19502.996} C_VEL
LIN {X 0,Y 237.575,Z 314.869,A -85,B 0,C 180,E1 -19505.173,E2 -19505.173} C_VEL
LIN {X 0,Y 239.952,Z 330.091,A -85,B 0,C 180,E1 -19505.891,E2 -19505.891} C_VEL
LIN {X 0,Y 243.304,Z 357.42,A -85,B 0,C 180,E1 -19507.066,E2 -19507.066} C_VEL
LIN {X 0,Y 242.291,Z 391.737,A -85,B 0,C 180,E1 -19508.156,E2 -19508.156} C_VEL
LIN {X 0,Y 241.655,Z 401.047,A -85,B 0,C 180,E1 -19508.64,E2 -19508.64} C_VEL
LIN {X 0,Y 240.777,Z 410.898,A -85,B 0,C 180,E1 -19509.392,E2 -19509.392} C_VEL
LIN {X 0,Y 239.681,Z 421.488,A -85,B 0,C 180,E1 -19510.517,E2 -19510.517} C_VEL
LIN {X 0,Y 238.283,Z 431.475,A -85,B 0,C 180,E1 -19511.96,E2 -19511.96} C_VEL
LIN {X 0,Y 237.143,Z 439.484,A -85,B 0,C 180,E1 -19513.427,E2 -19513.427} C_VEL
LIN {X 0,Y 236.068,Z 446.092,A -85,B 0,C 180,E1 -19514.901,E2 -19514.901} C_VEL
LIN {X 0,Y 235.106,Z 452.379,A -85,B 0,C 180,E1 -19516.605,E2 -19516.605} C_VEL
LIN {X 0,Y 234.281,Z 457.587,A -85,B 0,C 180,E1 -19518.318,E2 -19518.318} C_VEL
LIN {X 0,Y 233.809,Z 460.952,A -85,B 0,C 180,E1 -19519.61,E2 -19519.61} C_VEL
LIN {X 0,Y 233.3,Z 464.732,A -85,B 0,C 180,E1 -19521.337,E2 -19521.337} C_VEL
LIN {X 0,Y 232.841,Z 469.015,A -85,B 0,C 180,E1 -19523.936,E2 -19523.936} C_VEL
LIN {X 0,Y 232.758,Z 470.632,A -85,B 0,C 180,E1 -19525.147,E2 -19525.147} C_VEL
LIN {X 0,Y 232.755,Z 473.311,A -85,B 0,C 180,E1 -19528.27,E2 -19528.27} C_VEL
LIN {X 0,Y 232.82,Z 474.132,A -85,B 0,C 180,E1 -19530,E2 -19530} C_VEL
LIN {X 0,Y 232.733,Z 474.418,A -85,B 0,C 180,E1 -19531.73,E2 -19531.73} C_VEL
LIN {X 0,Y 232.72,Z 473.62,A -85,B 0,C 180,E1 -19534.744,E2 -19534.744} C_VEL
LIN {X 0,Y 233.004,Z 472.123,A -85,B 0,C 180,E1 -19536.929,E2 -19536.929} C_VEL
LIN {X 0,Y 233.665,Z 469.226,A -85,B 0,C 180,E1 -19539.522,E2 -19539.522} C_VEL
LIN {X 0,Y 234.725,Z 465.075,A -85,B 0,C 180,E1 -19542.098,E2 -19542.098} C_VEL
LIN {X 0,Y 236.286,Z 459.477,A -85,B 0,C 180,E1 -19544.644,E2 -19544.644} C_VEL
LIN {X 0,Y 237.858,Z 453.368,A -85,B 0,C 180,E1 -19546.743,E2 -19546.743} C_VEL
LIN {X 0,Y 239.368,Z 447.443,A -85,B 0,C 180,E1 -19548.398,E2 -19548.398} C_VEL
LIN {X 0,Y 241.151,Z 440.247,A -85,B 0,C 180,E1 -19550.025,E2 -19550.025} C_VEL
LIN {X 0,Y 242.853,Z 432.595,A -85,B 0,C 180,E1 -19551.429,E2 -19551.429} C_VEL
LIN {X 0,Y 244.5,Z 424.581,A -85,B 0,C 180,E1 -19552.609,E2 -19552.609} C_VEL
LIN {X 0,Y 245.796,Z 416.345,A -85,B 0,C 180,E1 -19553.596,E2 -19553.596} C_VEL
LIN {X 0,Y 247.03,Z 408.071,A -85,B 0,C 180,E1 -19554.355,E2 -19554.355} C_VEL
LIN {X 0,Y 248.181,Z 398.248,A -85,B 0,C 180,E1 -19555.018,E2 -19555.018} C_VEL
LIN {X 0,Y 248.958,Z 387.451,A -85,B 0,C 180,E1 -19555.501,E2 -19555.501} C_VEL
LIN {X 0,Y 249.99,Z 359.465,A -85,B 0,C 180,E1 -19556.354,E2 -19556.354} C_VEL
LIN {X 0,Y 247.896,Z 343.533,A -85,B 0,C 180,E1 -19557.219,E2 -19557.219} C_VEL
LIN {X 0,Y 245.389,Z 330.266,A -85,B 0,C 180,E1 -19558.072,E2 -19558.072} C_VEL
LIN {X 0,Y 239.485,Z 316.923,A -85,B 0,C 180,E1 -19559.52,E2 -19559.52} C_VEL
LIN {X 0,Y 237.744,Z 312.955,A -85,B 0,C 180,E1 -19560.021,E2 -19560.021} C_VEL
LIN {X 0,Y 235.731,Z 304.124,A -85,B 0,C 180,E1 -19564.502,E2 -19564.502} C_VEL
LIN {X 0,Y 234.921,Z 301.038,A -85,B 0,C 180,E1 -19566.27,E2 -19566.27} C_VEL
LIN {X 0,Y 234.939,Z 301.037,A -85,B 0,C 180,E1 -19568.944,E2 -19568.944} C_VEL
LIN {X 0,Y 234.874,Z 301.05,A -85,B 0,C 180,E1 -19573.487,E2 -19573.487} C_VEL
LIN {X 0,Y 234.874,Z 301.044,A -85,B 0,C 180,E1 -19576.511,E2 -19576.511} C_VEL
LIN {X 0,Y 234.915,Z 301.037,A -85,B 0,C 180,E1 -19581.078,E2 -19581.078} C_VEL
LIN {X 0,Y 234.928,Z 301.035,A -85,B 0,C 180,E1 -19585.362,E2 -19585.362} C_VEL
LIN {X 0,Y 234.926,Z 301.032,A -85,B 0,C 180,E1 -19589.432,E2 -19589.432} C_VEL
LIN {X 0,Y 234.988,Z 301.015,A -85,B 0,C 180,E1 -19593.793,E2 -19593.793} C_VEL
LIN {X 0,Y 234.991,Z 301.011,A -85,B 0,C 180,E1 -19598.968,E2 -19598.968} C_VEL
LIN {X 0,Y 235.09,Z 301.004,A -85,B 0,C 180,E1 -19603.059,E2 -19603.059} C_VEL
LIN {X 0,Y 235.106,Z 301.011,A -85,B 0,C 180,E1 -19607.922,E2 -19607.922} C_VEL
LIN {X 0,Y 235.324,Z 300.967,A -85,B 0,C 180,E1 -19611.412,E2 -19611.412} C_VEL
LIN {X 0,Y 235.384,Z 300.975,A -85,B 0,C 180,E1 -19613.141,E2 -19613.141} C_VEL
LIN {X 0,Y 235.586,Z 300.943,A -85,B 0,C 180,E1 -19618.291,E2 -19618.291} C_VEL
LIN {X 0,Y 235.586,Z 300.936,A -85,B 0,C 180,E1 -19621.71,E2 -19621.71} C_VEL
LIN {X 0,Y 235.344,Z 300.971,A -85,B 0,C 180,E1 -19626.861,E2 -19626.861} C_VEL
LIN {X 0,Y 235.208,Z 300.999,A -85,B 0,C 180,E1 -19630.328,E2 -19630.328} C_VEL
LIN {X 0,Y 235.101,Z 301.009,A -85,B 0,C 180,E1 -19635.608,E2 -19635.608} C_VEL
LIN {X 0,Y 235.001,Z 301.028,A -85,B 0,C 180,E1 -19639.206,E2 -19639.206} C_VEL
LIN {X 0,Y 234.955,Z 301.033,A -85,B 0,C 180,E1 -19642.884,E2 -19642.884} C_VEL
LIN {X 0,Y 234.963,Z 301.027,A -85,B 0,C 180,E1 -19646.658,E2 -19646.658} C_VEL
LIN {X 0,Y 234.913,Z 301.041,A -85,B 0,C 180,E1 -19650.695,E2 -19650.695} C_VEL
LIN {X 0,Y 235.43,Z 302.938,A -85,B 0,C 180,E1 -19651.682,E2 -19651.682} C_VEL
LIN {X 0,Y 237.457,Z 306.729,A -85,B 0,C 180,E1 -19652.191,E2 -19652.191} C_VEL
LIN {X 0,Y 243.536,Z 318.591,A -85,B 0,C 180,E1 -19653.653,E2 -19653.653} C_VEL
LIN {X 0,Y 248.567,Z 330.104,A -85,B 0,C 180,E1 -19654.846,E2 -19654.846} C_VEL
LIN {X 0,Y 250.483,Z 335.525,A -85,B 0,C 180,E1 -19655.315,E2 -19655.315} C_VEL
LIN {X 0,Y 250.774,Z 338.644,A -85,B 0,C 180,E1 -19655.467,E2 -19655.467} C_VEL
LIN {X 0,Y 249.02,Z 379.206,A -85,B 0,C 180,E1 -19656.711,E2 -19656.711} C_VEL
LIN {X 0,Y 248.279,Z 389.316,A -85,B 0,C 180,E1 -19657.235,E2 -19657.235} C_VEL
LIN {X 0,Y 247.126,Z 400.425,A -85,B 0,C 180,E1 -19658.103,E2 -19658.103} C_VEL
LIN {X 0,Y 245.715,Z 409.837,A -85,B 0,C 180,E1 -19659.126,E2 -19659.126} C_VEL
LIN {X 0,Y 244.191,Z 418.228,A -85,B 0,C 180,E1 -19660.3,E2 -19660.3} C_VEL
LIN {X 0,Y 242.432,Z 426.788,A -85,B 0,C 180,E1 -19661.818,E2 -19661.818} C_VEL
LIN {X 0,Y 240.911,Z 433.069,A -85,B 0,C 180,E1 -19663.173,E2 -19663.173} C_VEL
LIN {X 0,Y 239.294,Z 439.335,A -85,B 0,C 180,E1 -19664.82,E2 -19664.82} C_VEL
LIN {X 0,Y 237.814,Z 444.85,A -85,B 0,C 180,E1 -19666.601,E2 -19666.601} C_VEL
LIN {X 0,Y 236.501,Z 449.562,A -85,B 0,C 180,E1 -19668.479,E2 -19668.479} C_VEL
LIN {X 0,Y 235.022,Z 454.654,A -85,B 0,C 180,E1 -19671.101,E2 -19671.101} C_VEL
LIN {X 0,Y 234.046,Z 457.473,A -85,B 0,C 180,E1 -19673.091,E2 -19673.091} C_VEL
LIN {X 0,Y 233.465,Z 459.532,A -85,B 0,C 180,E1 -19675.114,E2 -19675.114} C_VEL
LIN {X 0,Y 232.864,Z 461.164,A -85,B 0,C 180,E1 -19677.679,E2 -19677.679} C_VEL
LIN {X 0,Y 232.612,Z 461.508,A -85,B 0,C 180,E1 -19679.095,E2 -19679.095} C_VEL
LIN {X 0,Y 232.426,Z 461.471,A -85,B 0,C 180,E1 -19681.27,E2 -19681.27} C_VEL
LIN {X 0,Y 232.402,Z 460.885,A -85,B 0,C 180,E1 -19683.025,E2 -19683.025} C_VEL
LIN {X 0,Y 232.579,Z 459.57,A -85,B 0,C 180,E1 -19685.031,E2 -19685.031} C_VEL
LIN {X 0,Y 232.896,Z 457.717,A -85,B 0,C 180,E1 -19686.903,E2 -19686.903} C_VEL
LIN {X 0,Y 233.332,Z 454.773,A -85,B 0,C 180,E1 -19689.024,E2 -19689.024} C_VEL
LIN {X 0,Y 234.067,Z 449.789,A -85,B 0,C 180,E1 -19691.624,E2 -19691.624} C_VEL
LIN {X 0,Y 234.929,Z 444.115,A -85,B 0,C 180,E1 -19693.893,E2 -19693.893} C_VEL
LIN {X 0,Y 235.905,Z 438.207,A -85,B 0,C 180,E1 -19695.772,E2 -19695.772} C_VEL
LIN {X 0,Y 237.344,Z 429.191,A -85,B 0,C 180,E1 -19698.038,E2 -19698.038} C_VEL
LIN {X 0,Y 238.532,Z 421.13,A -85,B 0,C 180,E1 -19699.604,E2 -19699.604} C_VEL
LIN {X 0,Y 239.686,Z 412.606,A -85,B 0,C 180,E1 -19700.932,E2 -19700.932} C_VEL
LIN {X 0,Y 240.647,Z 404.087,A -85,B 0,C 180,E1 -19701.99,E2 -19701.99} C_VEL
LIN {X 0,Y 241.361,Z 395.64,A -85,B 0,C 180,E1 -19702.815,E2 -19702.815} C_VEL
LIN {X 0,Y 242.067,Z 386.073,A -85,B 0,C 180,E1 -19703.503,E2 -19703.503} C_VEL
LIN {X 0,Y 242.646,Z 374.68,A -85,B 0,C 180,E1 -19704.034,E2 -19704.034} C_VEL
LIN {X 0,Y 243.696,Z 333.557,A -85,B 0,C 180,E1 -19705.296,E2 -19705.296} C_VEL
LIN {X 0,Y 241.169,Z 319.294,A -85,B 0,C 180,E1 -19705.979,E2 -19705.979} C_VEL
LIN {X 0,Y 235.678,Z 302.41,A -85,B 0,C 180,E1 -19707.062,E2 -19707.062} C_VEL
LIN {X 0,Y 235.533,Z 300.965,A -85,B 0,C 180,E1 -19707.863,E2 -19707.863} C_VEL
LIN {X 0,Y 235.658,Z 300.946,A -85,B 0,C 180,E1 -19710,E2 -19710} C_VEL
LIN {X 0,Y 235.597,Z 300.953,A -85,B 0,C 180,E1 -19711.709,E2 -19711.709} C_VEL
LIN {X 0,Y 235.362,Z 300.977,A -85,B 0,C 180,E1 -19716.86,E2 -19716.86} C_VEL
LIN {X 0,Y 235.216,Z 300.996,A -85,B 0,C 180,E1 -19720.327,E2 -19720.327} C_VEL
LIN {X 0,Y 235.087,Z 301.012,A -85,B 0,C 180,E1 -19725.608,E2 -19725.608} C_VEL
LIN {X 0,Y 234.99,Z 301.018,A -85,B 0,C 180,E1 -19729.207,E2 -19729.207} C_VEL
LIN {X 0,Y 234.952,Z 301.019,A -85,B 0,C 180,E1 -19732.883,E2 -19732.883} C_VEL
LIN {X 0,Y 234.969,Z 301.03,A -85,B 0,C 180,E1 -19736.657,E2 -19736.657} C_VEL
LIN {X 0,Y 234.931,Z 301.034,A -85,B 0,C 180,E1 -19740.567,E2 -19740.567} C_VEL
LIN {X 0,Y 234.926,Z 301.031,A -85,B 0,C 180,E1 -19744.638,E2 -19744.638} C_VEL
LIN {X 0,Y 234.94,Z 301.032,A -85,B 0,C 180,E1 -19748.943,E2 -19748.943} C_VEL
LIN {X 0,Y 234.894,Z 301.031,A -85,B 0,C 180,E1 -19753.483,E2 -19753.483} C_VEL
LIN {X 0,Y 234.962,Z 301.026,A -85,B 0,C 180,E1 -19756.531,E2 -19756.531} C_VEL
LIN {X 0,Y 234.952,Z 301.027,A -85,B 0,C 180,E1 -19761.085,E2 -19761.085} C_VEL
LIN {X 0,Y 234.957,Z 301.016,A -85,B 0,C 180,E1 -19765.366,E2 -19765.366} C_VEL
LIN {X 0,Y 234.964,Z 301.03,A -85,B 0,C 180,E1 -19770.157,E2 -19770.157} C_VEL
LIN {X 0,Y 234.989,Z 301.025,A -85,B 0,C 180,E1 -19773.793,E2 -19773.793} C_VEL
LIN {X 0,Y 235.006,Z 301.006,A -85,B 0,C 180,E1 -19778.969,E2 -19778.969} C_VEL
LIN {X 0,Y 235.091,Z 301.009,A -85,B 0,C 180,E1 -19783.059,E2 -19783.059} C_VEL
LIN {X 0,Y 235.107,Z 301.009,A -85,B 0,C 180,E1 -19787.921,E2 -19787.921} C_VEL
LIN {X 0,Y 235.324,Z 300.977,A -85,B 0,C 180,E1 -19791.412,E2 -19791.412} C_VEL
LIN {X 0,Y 235.366,Z 300.967,A -85,B 0,C 180,E1 -19793.14,E2 -19793.14} C_VEL
LIN {X 0,Y 235.587,Z 300.944,A -85,B 0,C 180,E1 -19798.29,E2 -19798.29} C_VEL
LIN {X 0,Y 235.588,Z 300.95,A -85,B 0,C 180,E1 -19801.709,E2 -19801.709} C_VEL
LIN {X 0,Y 235.365,Z 300.974,A -85,B 0,C 180,E1 -19806.86,E2 -19806.86} C_VEL
LIN {X 0,Y 235.208,Z 300.988,A -85,B 0,C 180,E1 -19810.328,E2 -19810.328} C_VEL
LIN {X 0,Y 235.1,Z 301.014,A -85,B 0,C 180,E1 -19815.607,E2 -19815.607} C_VEL
LIN {X 0,Y 234.999,Z 301.021,A -85,B 0,C 180,E1 -19819.206,E2 -19819.206} C_VEL
LIN {X 0,Y 234.946,Z 301.025,A -85,B 0,C 180,E1 -19822.884,E2 -19822.884} C_VEL
LIN {X 0,Y 234.961,Z 301.028,A -85,B 0,C 180,E1 -19826.658,E2 -19826.658} C_VEL
LIN {X 0,Y 234.916,Z 301.031,A -85,B 0,C 180,E1 -19830.57,E2 -19830.57} C_VEL
LIN {X 0,Y 234.925,Z 301.035,A -85,B 0,C 180,E1 -19834.639,E2 -19834.639} C_VEL
LIN {X 0,Y 234.881,Z 301.03,A -85,B 0,C 180,E1 -19837.496,E2 -19837.496} C_VEL
LIN {X 0,Y 234.19,Z 301.117,A -85,B 0,C 180,E1 -19838.928,E2 -19838.928} C_VEL
LIN {X 0,Y 231.331,Z 301.474,A -85,B 0,C 180,E1 -19841.263,E2 -19841.263} C_VEL
LIN {X 0,Y 228.925,Z 301.78,A -85,B 0,C 180,E1 -19843.168,E2 -19843.168} C_VEL
LIN {X 0,Y 227.907,Z 301.908,A -85,B 0,C 180,E1 -19844.646,E2 -19844.646} C_VEL
LIN {X 0,Y 227.831,Z 301.917,A -85,B 0,C 180,E1 -19845.147,E2 -19845.147} C_VEL
LIN {X 0,Y 227.823,Z 301.917,A -85,B 0,C 180,E1 -19849.624,E2 -19849.624} C_VEL
LIN {X 0,Y 227.877,Z 301.911,A -85,B 0,C 180,E1 -19854.129,E2 -19854.129} C_VEL
LIN {X 0,Y 227.964,Z 302.078,A -85,B 0,C 180,E1 -19858.662,E2 -19858.662} C_VEL
LIN {X 0,Y 229.574,Z 310.48,A -85,B 0,C 180,E1 -19862.665,E2 -19862.665} C_VEL
LIN {X 0,Y 230.311,Z 314.481,A -85,B 0,C 180,E1 -19864.498,E2 -19864.498} C_VEL
LIN {X 0,Y 231.774,Z 320.073,A -85,B 0,C 180,E1 -19864.828,E2 -19864.828} C_VEL
LIN {X 0,Y 236.331,Z 355.595,A -85,B 0,C 180,E1 -19866.444,E2 -19866.444} C_VEL
LIN {X 0,Y 236.508,Z 361.085,A -85,B 0,C 180,E1 -19866.643,E2 -19866.643} C_VEL
LIN {X 0,Y 235.513,Z 392.153,A -85,B 0,C 180,E1 -19867.667,E2 -19867.667} C_VEL
LIN {X 0,Y 234.781,Z 402.289,A -85,B 0,C 180,E1 -19868.229,E2 -19868.229} C_VEL
LIN {X 0,Y 233.832,Z 412.674,A -85,B 0,C 180,E1 -19869.09,E2 -19869.09} C_VEL
LIN {X 0,Y 232.537,Z 423.371,A -85,B 0,C 180,E1 -19870.353,E2 -19870.353} C_VEL
LIN {X 0,Y 231.321,Z 431.737,A -85,B 0,C 180,E1 -19871.627,E2 -19871.627} C_VEL
LIN {X 0,Y 230.148,Z 439.67,A -85,B 0,C 180,E1 -19873.137,E2 -19873.137} C_VEL
LIN {X 0,Y 228.915,Z 447.078,A -85,B 0,C 180,E1 -19874.873,E2 -19874.873} C_VEL
LIN {X 0,Y 227.726,Z 454.591,A -85,B 0,C 180,E1 -19877.071,E2 -19877.071} C_VEL
LIN {X 0,Y 226.808,Z 460.454,A -85,B 0,C 180,E1 -19879.286,E2 -19879.286} C_VEL
LIN {X 0,Y 226.275,Z 464.28,A -85,B 0,C 180,E1 -19881.066,E2 -19881.066} C_VEL
LIN {X 0,Y 225.777,Z 468.639,A -85,B 0,C 180,E1 -19883.745,E2 -19883.745} C_VEL
LIN {X 0,Y 225.665,Z 470.59,A -85,B 0,C 180,E1 -19885.266,E2 -19885.266} C_VEL
LIN {X 0,Y 225.67,Z 473.039,A -85,B 0,C 180,E1 -19888.215,E2 -19888.215} C_VEL
LIN {X 0,Y 225.731,Z 473.909,A -85,B 0,C 180,E1 -19890,E2 -19890} C_VEL
LIN {X 0,Y 225.649,Z 474.201,A -85,B 0,C 180,E1 -19891.785,E2 -19891.785} C_VEL
LIN {X 0,Y 225.612,Z 473.674,A -85,B 0,C 180,E1 -19894.568,E2 -19894.568} C_VEL
LIN {X 0,Y 225.944,Z 472.047,A -85,B 0,C 180,E1 -19897.147,E2 -19897.147} C_VEL
LIN {X 0,Y 226.665,Z 469.204,A -85,B 0,C 180,E1 -19899.818,E2 -19899.818} C_VEL
LIN {X 0,Y 227.779,Z 465.118,A -85,B 0,C 180,E1 -19902.473,E2 -19902.473} C_VEL
LIN {X 0,Y 229.429,Z 459.63,A -85,B 0,C 180,E1 -19905.092,E2 -19905.092} C_VEL
LIN {X 0,Y 231.088,Z 453.65,A -85,B 0,C 180,E1 -19907.248,E2 -19907.248} C_VEL
LIN {X 0,Y 233.096,Z 446.117,A -85,B 0,C 180,E1 -19909.369,E2 -19909.369} C_VEL
LIN {X 0,Y 234.789,Z 439.715,A -85,B 0,C 180,E1 -19910.821,E2 -19910.821} C_VEL
LIN {X 0,Y 236.576,Z 431.995,A -85,B 0,C 180,E1 -19912.257,E2 -19912.257} C_VEL
LIN {X 0,Y 238.24,Z 423.902,A -85,B 0,C 180,E1 -19913.468,E2 -19913.468} C_VEL
LIN {X 0,Y 239.588,Z 415.986,A -85,B 0,C 180,E1 -19914.421,E2 -19914.421} C_VEL
LIN {X 0,Y 241.016,Z 406.8,A -85,B 0,C 180,E1 -19915.263,E2 -19915.263} C_VEL
LIN {X 0,Y 242.299,Z 395.884,A -85,B 0,C 180,E1 -19915.979,E2 -19915.979} C_VEL
LIN {X 0,Y 243.145,Z 381.747,A -85,B 0,C 180,E1 -19916.513,E2 -19916.513} C_VEL
LIN {X 0,Y 243.835,Z 359.772,A -85,B 0,C 180,E1 -19917.217,E2 -19917.217} C_VEL
LIN {X 0,Y 241.835,Z 344.261,A -85,B 0,C 180,E1 -19918.098,E2 -19918.098} C_VEL
LIN {X 0,Y 239.55,Z 332.603,A -85,B 0,C 180,E1 -19918.907,E2 -19918.907} C_VEL
LIN {X 0,Y 233.839,Z 319.957,A -85,B 0,C 180,E1 -19920.369,E2 -19920.369} C_VEL
LIN {X 0,Y 231.86,Z 315.968,A -85,B 0,C 180,E1 -19920.888,E2 -19920.888} C_VEL
LIN {X 0,Y 230.464,Z 312.731,A -85,B 0,C 180,E1 -19921.319,E2 -19921.319} C_VEL
LIN {X 0,Y 229.014,Z 306.274,A -85,B 0,C 180,E1 -19924.744,E2 -19924.744} C_VEL
LIN {X 0,Y 227.861,Z 301.916,A -85,B 0,C 180,E1 -19927.312,E2 -19927.312} C_VEL
LIN {X 0,Y 227.821,Z 301.928,A -85,B 0,C 180,E1 -19930.376,E2 -19930.376} C_VEL
LIN {X 0,Y 227.821,Z 301.918,A -85,B 0,C 180,E1 -19935.194,E2 -19935.194} C_VEL
LIN {X 0,Y 227.82,Z 301.915,A -85,B 0,C 180,E1 -19939.622,E2 -19939.622} C_VEL
LIN {X 0,Y 227.877,Z 301.908,A -85,B 0,C 180,E1 -19944.128,E2 -19944.128} C_VEL
LIN {X 0,Y 227.865,Z 301.904,A -85,B 0,C 180,E1 -19948.377,E2 -19948.377} C_VEL
LIN {X 0,Y 227.88,Z 301.895,A -85,B 0,C 180,E1 -19952.444,E2 -19952.444} C_VEL
LIN {X 0,Y 227.9,Z 301.904,A -85,B 0,C 180,E1 -19956.366,E2 -19956.366} C_VEL
LIN {X 0,Y 227.931,Z 301.899,A -85,B 0,C 180,E1 -19960.174,E2 -19960.174} C_VEL
LIN {X 0,Y 228.05,Z 301.873,A -85,B 0,C 180,E1 -19963.897,E2 -19963.897} C_VEL
LIN {X 0,Y 228.064,Z 301.888,A -85,B 0,C 180,E1 -19967.543,E2 -19967.543} C_VEL
LIN {X 0,Y 228.26,Z 301.845,A -85,B 0,C 180,E1 -19971.144,E2 -19971.144} C_VEL
LIN {X 0,Y 228.331,Z 301.851,A -85,B 0,C 180,E1 -19972.928,E2 -19972.928} C_VEL
LIN {X 0,Y 228.545,Z 301.819,A -85,B 0,C 180,E1 -19978.238,E2 -19978.238} C_VEL
LIN {X 0,Y 228.544,Z 301.812,A -85,B 0,C 180,E1 -19981.762,E2 -19981.762} C_VEL
LIN {X 0,Y 228.296,Z 301.848,A -85,B 0,C 180,E1 -19987.073,E2 -19987.073} C_VEL
LIN {X 0,Y 228.139,Z 301.88,A -85,B 0,C 180,E1 -19990.652,E2 -19990.652} C_VEL
LIN {X 0,Y 228.053,Z 301.891,A -85,B 0,C 180,E1 -19994.273,E2 -19994.273} C_VEL
LIN {X 0,Y 227.997,Z 301.896,A -85,B 0,C 180,E1 -19997.954,E2 -19997.954} C_VEL
LIN {X 0,Y 227.925,Z 301.911,A -85,B 0,C 180,E1 -20002.33,E2 -20002.33} C_VEL
LIN {X 0,Y 227.937,Z 301.902,A -85,B 0,C 180,E1 -20006.603,E2 -20006.603} C_VEL
LIN {X 0,Y 227.902,Z 302.006,A -85,B 0,C 180,E1 -20009.704,E2 -20009.704} C_VEL
LIN {X 0,Y 228.239,Z 303.382,A -85,B 0,C 180,E1 -20010.351,E2 -20010.351} C_VEL
LIN {X 0,Y 230.473,Z 307.287,A -85,B 0,C 180,E1 -20010.947,E2 -20010.947} C_VEL
LIN {X 0,Y 236.866,Z 319.399,A -85,B 0,C 180,E1 -20012.586,E2 -20012.586} C_VEL
LIN {X 0,Y 241.834,Z 330.357,A -85,B 0,C 180,E1 -20013.827,E2 -20013.827} C_VEL
LIN {X 0,Y 244.633,Z 337.732,A -85,B 0,C 180,E1 -20014.541,E2 -20014.541} C_VEL
LIN {X 0,Y 242.881,Z 379.757,A -85,B 0,C 180,E1 -20015.886,E2 -20015.886} C_VEL
LIN {X 0,Y 242.108,Z 389.837,A -85,B 0,C 180,E1 -20016.428,E2 -20016.428} C_VEL
LIN {X 0,Y 240.863,Z 401.078,A -85,B 0,C 180,E1 -20017.337,E2 -20017.337} C_VEL
LIN {X 0,Y 239.197,Z 411.455,A -85,B 0,C 180,E1 -20018.532,E2 -20018.532} C_VEL
LIN {X 0,Y 237.601,Z 419.603,A -85,B 0,C 180,E1 -20019.733,E2 -20019.733} C_VEL
LIN {X 0,Y 236.23,Z 425.992,A -85,B 0,C 180,E1 -20020.883,E2 -20020.883} C_VEL
LIN {X 0,Y 234.748,Z 432.096,A -85,B 0,C 180,E1 -20022.187,E2 -20022.187} C_VEL
LIN {X 0,Y 232.921,Z 438.819,A -85,B 0,C 180,E1 -20023.947,E2 -20023.947} C_VEL
LIN {X 0,Y 231.339,Z 444.219,A -85,B 0,C 180,E1 -20025.676,E2 -20025.676} C_VEL
LIN {X 0,Y 229.869,Z 449.355,A -85,B 0,C 180,E1 -20027.732,E2 -20027.732} C_VEL
LIN {X 0,Y 228.584,Z 453.436,A -85,B 0,C 180,E1 -20029.786,E2 -20029.786} C_VEL
LIN {X 0,Y 227.55,Z 456.614,A -85,B 0,C 180,E1 -20031.852,E2 -20031.852} C_VEL
LIN {X 0,Y 226.697,Z 458.981,A -85,B 0,C 180,E1 -20033.913,E2 -20033.913} C_VEL
LIN {X 0,Y 225.877,Z 461.229,A -85,B 0,C 180,E1 -20037.15,E2 -20037.15} C_VEL
LIN {X 0,Y 225.41,Z 461.861,A -85,B 0,C 180,E1 -20040.077,E2 -20040.077} C_VEL
LIN {X 0,Y 225.309,Z 461.472,A -85,B 0,C 180,E1 -20042.104,E2 -20042.104} C_VEL
LIN {X 0,Y 225.436,Z 460.031,A -85,B 0,C 180,E1 -20044.7,E2 -20044.7} C_VEL
LIN {X 0,Y 225.85,Z 457.67,A -85,B 0,C 180,E1 -20047.11,E2 -20047.11} C_VEL
LIN {X 0,Y 226.312,Z 454.447,A -85,B 0,C 180,E1 -20049.411,E2 -20049.411} C_VEL
LIN {X 0,Y 226.91,Z 450.631,A -85,B 0,C 180,E1 -20051.491,E2 -20051.491} C_VEL
LIN {X 0,Y 227.786,Z 444.973,A -85,B 0,C 180,E1 -20053.879,E2 -20053.879} C_VEL
LIN {X 0,Y 228.778,Z 439.336,A -85,B 0,C 180,E1 -20055.774,E2 -20055.774} C_VEL
LIN {X 0,Y 229.889,Z 432.508,A -85,B 0,C 180,E1 -20057.644,E2 -20057.644} C_VEL
LIN {X 0,Y 231.238,Z 424.121,A -85,B 0,C 180,E1 -20059.493,E2 -20059.493} C_VEL
LIN {X 0,Y 232.572,Z 414.768,A -85,B 0,C 180,E1 -20061.091,E2 -20061.091} C_VEL
LIN {X 0,Y 233.687,Z 405.795,A -85,B 0,C 180,E1 -20062.283,E2 -20062.283} C_VEL
LIN {X 0,Y 234.489,Z 396.914,A -85,B 0,C 180,E1 -20063.207,E2 -20063.207} C_VEL
LIN {X 0,Y 235.219,Z 387.684,A -85,B 0,C 180,E1 -20063.918,E2 -20063.918} C_VEL
LIN {X 0,Y 235.756,Z 378.773,A -85,B 0,C 180,E1 -20064.39,E2 -20064.39} C_VEL
LIN {X 0,Y 237.041,Z 334.751,A -85,B 0,C 180,E1 -20065.815,E2 -20065.815} C_VEL
LIN {X 0,Y 234.735,Z 321.481,A -85,B 0,C 180,E1 -20066.47,E2 -20066.47} C_VEL
LIN {X 0,Y 228.573,Z 302.58,A -85,B 0,C 180,E1 -20067.742,E2 -20067.742} C_VEL
LIN {X 0,Y 228.57,Z 301.831,A -85,B 0,C 180,E1 -20068.238,E2 -20068.238} C_VEL
LIN {X 0,Y 228.555,Z 301.83,A -85,B 0,C 180,E1 -20071.762,E2 -20071.762} C_VEL
LIN {X 0,Y 228.314,Z 301.855,A -85,B 0,C 180,E1 -20077.073,E2 -20077.073} C_VEL
LIN {X 0,Y 228.147,Z 301.874,A -85,B 0,C 180,E1 -20080.651,E2 -20080.651} C_VEL
LIN {X 0,Y 228.05,Z 301.887,A -85,B 0,C 180,E1 -20084.273,E2 -20084.273} C_VEL
LIN {X 0,Y 227.969,Z 301.898,A -85,B 0,C 180,E1 -20087.955,E2 -20087.955} C_VEL
LIN {X 0,Y 227.915,Z 301.889,A -85,B 0,C 180,E1 -20092.319,E2 -20092.319} C_VEL
LIN {X 0,Y 227.943,Z 301.904,A -85,B 0,C 180,E1 -20096.602,E2 -20096.602} C_VEL
LIN {X 0,Y 227.908,Z 301.908,A -85,B 0,C 180,E1 -20100.295,E2 -20100.295} C_VEL
LIN {X 0,Y 227.876,Z 301.908,A -85,B 0,C 180,E1 -20103.72,E2 -20103.72} C_VEL
LIN {X 0,Y 227.842,Z 301.915,A -85,B 0,C 180,E1 -20108.09,E2 -20108.09} C_VEL
LIN {X 0,Y 227.815,Z 301.908,A -85,B 0,C 180,E1 -20112.74,E2 -20112.74} C_VEL
LIN {X 0,Y 227.906,Z 301.908,A -85,B 0,C 180,E1 -20117.279,E2 -20117.279} C_VEL
LIN {X 0,Y 227.868,Z 301.908,A -85,B 0,C 180,E1 -20121.913,E2 -20121.913} C_VEL
LIN {X 0,Y 227.887,Z 301.903,A -85,B 0,C 180,E1 -20126.372,E2 -20126.372} C_VEL
LIN {X 0,Y 227.914,Z 301.906,A -85,B 0,C 180,E1 -20130.437,E2 -20130.437} C_VEL
LIN {X 0,Y 227.924,Z 301.903,A -85,B 0,C 180,E1 -20134.425,E2 -20134.425} C_VEL
LIN {X 0,Y 227.957,Z 301.888,A -85,B 0,C 180,E1 -20138.286,E2 -20138.286} C_VEL
LIN {X 0,Y 228.029,Z 301.889,A -85,B 0,C 180,E1 -20142.826,E2 -20142.826} C_VEL
LIN {X 0,Y 228.065,Z 301.886,A -85,B 0,C 180,E1 -20147.543,E2 -20147.543} C_VEL
LIN {X 0,Y 228.261,Z 301.858,A -85,B 0,C 180,E1 -20151.144,E2 -20151.144} C_VEL
LIN {X 0,Y 228.316,Z 301.846,A -85,B 0,C 180,E1 -20152.927,E2 -20152.927} C_VEL
LIN {X 0,Y 228.546,Z 301.82,A -85,B 0,C 180,E1 -20158.238,E2 -20158.238} C_VEL
LIN {X 0,Y 228.546,Z 301.827,A -85,B 0,C 180,E1 -20161.762,E2 -20161.762} C_VEL
LIN {X 0,Y 228.316,Z 301.852,A -85,B 0,C 180,E1 -20167.072,E2 -20167.072} C_VEL
LIN {X 0,Y 228.139,Z 301.868,A -85,B 0,C 180,E1 -20170.651,E2 -20170.651} C_VEL
LIN {X 0,Y 228.053,Z 301.888,A -85,B 0,C 180,E1 -20174.273,E2 -20174.273} C_VEL
LIN {X 0,Y 227.996,Z 301.895,A -85,B 0,C 180,E1 -20177.954,E2 -20177.954} C_VEL
LIN {X 0,Y 227.911,Z 301.903,A -85,B 0,C 180,E1 -20182.321,E2 -20182.321} C_VEL
LIN {X 0,Y 227.936,Z 301.903,A -85,B 0,C 180,E1 -20186.602,E2 -20186.602} C_VEL
LIN {X 0,Y 227.891,Z 301.906,A -85,B 0,C 180,E1 -20190.291,E2 -20190.291} C_VEL
LIN {X 0,Y 227.872,Z 301.912,A -85,B 0,C 180,E1 -20193.721,E2 -20193.721} C_VEL
LIN {X 0,Y 227.839,Z 301.914,A -85,B 0,C 180,E1 -20198.092,E2 -20198.092} C_VEL
LIN {X 0,Y 227.808,Z 301.912,A -85,B 0,C 180,E1 -20202.743,E2 -20202.743} C_VEL
LIN {X 0,Y 227.831,Z 301.917,A -85,B 0,C 180,E1 -20205.147,E2 -20205.147} C_VEL
LIN {X 0,Y 227.198,Z 301.998,A -85,B 0,C 180,E1 -20206.623,E2 -20206.623} C_VEL
LIN {X 0,Y 224.411,Z 302.349,A -85,B 0,C 180,E1 -20209.034,E2 -20209.034} C_VEL
LIN {X 0,Y 221.166,Z 302.751,A -85,B 0,C 180,E1 -20212.012,E2 -20212.012} C_VEL
LIN {X 0,Y 220.802,Z 302.791,A -85,B 0,C 180,E1 -20213.043,E2 -20213.043} C_VEL
LIN {X 0,Y 220.873,Z 302.901,A -85,B 0,C 180,E1 -20218.248,E2 -20218.248} C_VEL
LIN {X 0,Y 222.299,Z 309.876,A -85,B 0,C 180,E1 -20221.692,E2 -20221.692} C_VEL
LIN {X 0,Y 223.028,Z 314.206,A -85,B 0,C 180,E1 -20223.765,E2 -20223.765} C_VEL
LIN {X 0,Y 225.153,Z 321.26,A -85,B 0,C 180,E1 -20224.243,E2 -20224.243} C_VEL
LIN {X 0,Y 229.791,Z 357.676,A -85,B 0,C 180,E1 -20225.956,E2 -20225.956} C_VEL
LIN {X 0,Y 228.763,Z 391.672,A -85,B 0,C 180,E1 -20227.108,E2 -20227.108} C_VEL
LIN {X 0,Y 228.085,Z 401.309,A -85,B 0,C 180,E1 -20227.648,E2 -20227.648} C_VEL
LIN {X 0,Y 227.149,Z 411.016,A -85,B 0,C 180,E1 -20228.444,E2 -20228.444} C_VEL
LIN {X 0,Y 225.867,Z 422.234,A -85,B 0,C 180,E1 -20229.748,E2 -20229.748} C_VEL
LIN {X 0,Y 224.558,Z 430.763,A -85,B 0,C 180,E1 -20231.053,E2 -20231.053} C_VEL
LIN {X 0,Y 223.504,Z 437.799,A -85,B 0,C 180,E1 -20232.383,E2 -20232.383} C_VEL
LIN {X 0,Y 222.36,Z 444.625,A -85,B 0,C 180,E1 -20233.946,E2 -20233.946} C_VEL
LIN {X 0,Y 221.234,Z 451.087,A -85,B 0,C 180,E1 -20235.748,E2 -20235.748} C_VEL
LIN {X 0,Y 220.342,Z 456.454,A -85,B 0,C 180,E1 -20237.567,E2 -20237.567} C_VEL
LIN {X 0,Y 219.522,Z 461.891,A -85,B 0,C 180,E1 -20239.859,E2 -20239.859} C_VEL
LIN {X 0,Y 219.048,Z 465.401,A -85,B 0,C 180,E1 -20241.699,E2 -20241.699} C_VEL
LIN {X 0,Y 218.631,Z 469.424,A -85,B 0,C 180,E1 -20244.466,E2 -20244.466} C_VEL
LIN {X 0,Y 218.533,Z 471.355,A -85,B 0,C 180,E1 -20246.312,E2 -20246.312} C_VEL
LIN {X 0,Y 218.568,Z 472.767,A -85,B 0,C 180,E1 -20248.157,E2 -20248.157} C_VEL
LIN {X 0,Y 218.645,Z 473.674,A -85,B 0,C 180,E1 -20250,E2 -20250} C_VEL
LIN {X 0,Y 218.547,Z 473.977,A -85,B 0,C 180,E1 -20251.843,E2 -20251.843} C_VEL
LIN {X 0,Y 218.512,Z 473.634,A -85,B 0,C 180,E1 -20254.403,E2 -20254.403} C_VEL
LIN {X 0,Y 218.879,Z 471.986,A -85,B 0,C 180,E1 -20257.379,E2 -20257.379} C_VEL
LIN {X 0,Y 219.653,Z 469.204,A -85,B 0,C 180,E1 -20260.135,E2 -20260.135} C_VEL
LIN {X 0,Y 220.832,Z 465.179,A -85,B 0,C 180,E1 -20262.872,E2 -20262.872} C_VEL
LIN {X 0,Y 221.934,Z 461.705,A -85,B 0,C 180,E1 -20264.675,E2 -20264.675} C_VEL
LIN {X 0,Y 223.585,Z 456.341,A -85,B 0,C 180,E1 -20266.903,E2 -20266.903} C_VEL
LIN {X 0,Y 225.55,Z 449.666,A -85,B 0,C 180,E1 -20269.097,E2 -20269.097} C_VEL
LIN {X 0,Y 227.929,Z 441.223,A -85,B 0,C 180,E1 -20271.241,E2 -20271.241} C_VEL
LIN {X 0,Y 230.044,Z 432.622,A -85,B 0,C 180,E1 -20272.924,E2 -20272.924} C_VEL
LIN {X 0,Y 231.788,Z 424.726,A -85,B 0,C 180,E1 -20274.162,E2 -20274.162} C_VEL
LIN {X 0,Y 233.228,Z 416.878,A -85,B 0,C 180,E1 -20275.159,E2 -20275.159} C_VEL
LIN {X 0,Y 234.66,Z 408.291,A -85,B 0,C 180,E1 -20275.997,E2 -20275.997} C_VEL
LIN {X 0,Y 235.893,Z 398.748,A -85,B 0,C 180,E1 -20276.686,E2 -20276.686} C_VEL
LIN {X 0,Y 236.753,Z 388.505,A -85,B 0,C 180,E1 -20277.183,E2 -20277.183} C_VEL
LIN {X 0,Y 237.81,Z 360.407,A -85,B 0,C 180,E1 -20278.118,E2 -20278.118} C_VEL
LIN {X 0,Y 235.992,Z 346,A -85,B 0,C 180,E1 -20278.971,E2 -20278.971} C_VEL
LIN {X 0,Y 233.9,Z 335.261,A -85,B 0,C 180,E1 -20279.748,E2 -20279.748} C_VEL
LIN {X 0,Y 227.551,Z 321.13,A -85,B 0,C 180,E1 -20281.485,E2 -20281.485} C_VEL
LIN {X 0,Y 224.37,Z 315.222,A -85,B 0,C 180,E1 -20282.366,E2 -20282.366} C_VEL
LIN {X 0,Y 223.184,Z 312.43,A -85,B 0,C 180,E1 -20282.781,E2 -20282.781} C_VEL
LIN {X 0,Y 221.598,Z 305.906,A -85,B 0,C 180,E1 -20286.486,E2 -20286.486} C_VEL
LIN {X 0,Y 220.808,Z 302.8,A -85,B 0,C 180,E1 -20288.434,E2 -20288.434} C_VEL
LIN {X 0,Y 220.757,Z 302.803,A -85,B 0,C 180,E1 -20292.927,E2 -20292.927} C_VEL
LIN {X 0,Y 220.757,Z 302.804,A -85,B 0,C 180,E1 -20297.071,E2 -20297.071} C_VEL
LIN {X 0,Y 220.802,Z 302.794,A -85,B 0,C 180,E1 -20300.462,E2 -20300.462} C_VEL
LIN {X 0,Y 220.797,Z 302.794,A -85,B 0,C 180,E1 -20305.045,E2 -20305.045} C_VEL
LIN {X 0,Y 220.863,Z 302.783,A -85,B 0,C 180,E1 -20309.394,E2 -20309.394} C_VEL
LIN {X 0,Y 220.889,Z 302.769,A -85,B 0,C 180,E1 -20313.549,E2 -20313.549} C_VEL
LIN {X 0,Y 220.859,Z 302.771,A -85,B 0,C 180,E1 -20317.552,E2 -20317.552} C_VEL
LIN {X 0,Y 220.978,Z 302.765,A -85,B 0,C 180,E1 -20322.571,E2 -20322.571} C_VEL
LIN {X 0,Y 221.004,Z 302.768,A -85,B 0,C 180,E1 -20327.138,E2 -20327.138} C_VEL
LIN {X 0,Y 221.198,Z 302.724,A -85,B 0,C 180,E1 -20330.859,E2 -20330.859} C_VEL
LIN {X 0,Y 221.264,Z 302.728,A -85,B 0,C 180,E1 -20332.701,E2 -20332.701} C_VEL
LIN {X 0,Y 221.503,Z 302.695,A -85,B 0,C 180,E1 -20338.182,E2 -20338.182} C_VEL
LIN {X 0,Y 221.502,Z 302.689,A -85,B 0,C 180,E1 -20341.818,E2 -20341.818} C_VEL
LIN {X 0,Y 221.233,Z 302.726,A -85,B 0,C 180,E1 -20347.301,E2 -20347.301} C_VEL
LIN {X 0,Y 221.061,Z 302.758,A -85,B 0,C 180,E1 -20350.997,E2 -20350.997} C_VEL
LIN {X 0,Y 221.008,Z 302.76,A -85,B 0,C 180,E1 -20356.631,E2 -20356.631} C_VEL
LIN {X 0,Y 220.886,Z 302.779,A -85,B 0,C 180,E1 -20360.487,E2 -20360.487} C_VEL
LIN {X 0,Y 220.862,Z 302.786,A -85,B 0,C 180,E1 -20364.436,E2 -20364.436} C_VEL
LIN {X 0,Y 220.819,Z 302.806,A -85,B 0,C 180,E1 -20368.516,E2 -20368.516} C_VEL
LIN {X 0,Y 220.907,Z 303.334,A -85,B 0,C 180,E1 -20368.828,E2 -20368.828} C_VEL
LIN {X 0,Y 222.166,Z 306.12,A -85,B 0,C 180,E1 -20369.232,E2 -20369.232} C_VEL
LIN {X 0,Y 223.726,Z 308.289,A -85,B 0,C 180,E1 -20369.654,E2 -20369.654} C_VEL
LIN {X 0,Y 230.214,Z 320.172,A -85,B 0,C 180,E1 -20371.432,E2 -20371.432} C_VEL
LIN {X 0,Y 236.148,Z 332.981,A -85,B 0,C 180,E1 -20372.997,E2 -20372.997} C_VEL
LIN {X 0,Y 238.728,Z 339.573,A -85,B 0,C 180,E1 -20373.68,E2 -20373.68} C_VEL
LIN {X 0,Y 236.855,Z 380.202,A -85,B 0,C 180,E1 -20375.002,E2 -20375.002} C_VEL
LIN {X 0,Y 235.919,Z 391.144,A -85,B 0,C 180,E1 -20375.611,E2 -20375.611} C_VEL
LIN {X 0,Y 234.502,Z 402.81,A -85,B 0,C 180,E1 -20376.642,E2 -20376.642} C_VEL
LIN {X 0,Y 232.918,Z 411.94,A -85,B 0,C 180,E1 -20377.735,E2 -20377.735} C_VEL
LIN {X 0,Y 231.402,Z 419.383,A -85,B 0,C 180,E1 -20378.854,E2 -20378.854} C_VEL
LIN {X 0,Y 229.527,Z 427.554,A -85,B 0,C 180,E1 -20380.391,E2 -20380.391} C_VEL
LIN {X 0,Y 228.064,Z 433.103,A -85,B 0,C 180,E1 -20381.646,E2 -20381.646} C_VEL
LIN {X 0,Y 226.574,Z 438.334,A -85,B 0,C 180,E1 -20383.032,E2 -20383.032} C_VEL
LIN {X 0,Y 224.509,Z 444.973,A -85,B 0,C 180,E1 -20385.227,E2 -20385.227} C_VEL
LIN {X 0,Y 222.991,Z 450.008,A -85,B 0,C 180,E1 -20387.344,E2 -20387.344} C_VEL
LIN {X 0,Y 222.231,Z 452.193,A -85,B 0,C 180,E1 -20388.387,E2 -20388.387} C_VEL
LIN {X 0,Y 221.07,Z 455.726,A -85,B 0,C 180,E1 -20390.521,E2 -20390.521} C_VEL
LIN {X 0,Y 219.887,Z 458.79,A -85,B 0,C 180,E1 -20393.04,E2 -20393.04} C_VEL
LIN {X 0,Y 219.343,Z 460.294,A -85,B 0,C 180,E1 -20394.78,E2 -20394.78} C_VEL
LIN {X 0,Y 218.822,Z 461.47,A -85,B 0,C 180,E1 -20396.908,E2 -20396.908} C_VEL
LIN {X 0,Y 218.298,Z 461.976,A -85,B 0,C 180,E1 -20400.372,E2 -20400.372} C_VEL
LIN {X 0,Y 218.296,Z 460.437,A -85,B 0,C 180,E1 -20404.351,E2 -20404.351} C_VEL
LIN {X 0,Y 218.801,Z 457.609,A -85,B 0,C 180,E1 -20407.329,E2 -20407.329} C_VEL
LIN {X 0,Y 219.187,Z 454.903,A -85,B 0,C 180,E1 -20409.348,E2 -20409.348} C_VEL
LIN {X 0,Y 219.922,Z 450.43,A -85,B 0,C 180,E1 -20411.836,E2 -20411.836} C_VEL
LIN {X 0,Y 220.623,Z 445.943,A -85,B 0,C 180,E1 -20413.816,E2 -20413.816} C_VEL
LIN {X 0,Y 221.617,Z 440.467,A -85,B 0,C 180,E1 -20415.773,E2 -20415.773} C_VEL
LIN {X 0,Y 222.707,Z 434.092,A -85,B 0,C 180,E1 -20417.632,E2 -20417.632} C_VEL
LIN {X 0,Y 223.94,Z 426.746,A -85,B 0,C 180,E1 -20419.376,E2 -20419.376} C_VEL
LIN {X 0,Y 225.083,Z 419.433,A -85,B 0,C 180,E1 -20420.792,E2 -20420.792} C_VEL
LIN {X 0,Y 226.309,Z 410.668,A -85,B 0,C 180,E1 -20422.164,E2 -20422.164} C_VEL
LIN {X 0,Y 227.495,Z 399.936,A -85,B 0,C 180,E1 -20423.459,E2 -20423.459} C_VEL
LIN {X 0,Y 228.407,Z 389.035,A -85,B 0,C 180,E1 -20424.372,E2 -20424.372} C_VEL
LIN {X 0,Y 228.978,Z 379.506,A -85,B 0,C 180,E1 -20424.913,E2 -20424.913} C_VEL
LIN {X 0,Y 230.338,Z 335.387,A -85,B 0,C 180,E1 -20426.388,E2 -20426.388} C_VEL
LIN {X 0,Y 228.252,Z 323.469,A -85,B 0,C 180,E1 -20426.995,E2 -20426.995} C_VEL
LIN {X 0,Y 221.544,Z 302.837,A -85,B 0,C 180,E1 -20428.409,E2 -20428.409} C_VEL
LIN {X 0,Y 221.513,Z 302.707,A -85,B 0,C 180,E1 -20431.818,E2 -20431.818} C_VEL
LIN {X 0,Y 221.25,Z 302.735,A -85,B 0,C 180,E1 -20437.3,E2 -20437.3} C_VEL
LIN {X 0,Y 221.068,Z 302.754,A -85,B 0,C 180,E1 -20440.996,E2 -20440.996} C_VEL
LIN {X 0,Y 220.992,Z 302.77,A -85,B 0,C 180,E1 -20446.631,E2 -20446.631} C_VEL
LIN {X 0,Y 220.871,Z 302.769,A -85,B 0,C 180,E1 -20450.488,E2 -20450.488} C_VEL
LIN {X 0,Y 220.862,Z 302.779,A -85,B 0,C 180,E1 -20454.435,E2 -20454.435} C_VEL
LIN {X 0,Y 220.836,Z 302.792,A -85,B 0,C 180,E1 -20458.513,E2 -20458.513} C_VEL
LIN {X 0,Y 220.817,Z 302.787,A -85,B 0,C 180,E1 -20462.755,E2 -20462.755} C_VEL
LIN {X 0,Y 220.809,Z 302.795,A -85,B 0,C 180,E1 -20467.277,E2 -20467.277} C_VEL
LIN {X 0,Y 220.772,Z 302.786,A -85,B 0,C 180,E1 -20471.951,E2 -20471.951} C_VEL
LIN {X 0,Y 220.864,Z 302.784,A -85,B 0,C 180,E1 -20477.042,E2 -20477.042} C_VEL
LIN {X 0,Y 220.853,Z 302.783,A -85,B 0,C 180,E1 -20480.473,E2 -20480.473} C_VEL
LIN {X 0,Y 220.812,Z 302.775,A -85,B 0,C 180,E1 -20485.047,E2 -20485.047} C_VEL
LIN {X 0,Y 220.864,Z 302.781,A -85,B 0,C 180,E1 -20489.394,E2 -20489.394} C_VEL
LIN {X 0,Y 220.89,Z 302.78,A -85,B 0,C 180,E1 -20493.549,E2 -20493.549} C_VEL
LIN {X 0,Y 220.873,Z 302.773,A -85,B 0,C 180,E1 -20497.553,E2 -20497.553} C_VEL
LIN {X 0,Y 220.979,Z 302.765,A -85,B 0,C 180,E1 -20502.571,E2 -20502.571} C_VEL
LIN {X 0,Y 221.004,Z 302.767,A -85,B 0,C 180,E1 -20507.138,E2 -20507.138} C_VEL
LIN {X 0,Y 221.198,Z 302.739,A -85,B 0,C 180,E1 -20510.859,E2 -20510.859} C_VEL
LIN {X 0,Y 221.252,Z 302.727,A -85,B 0,C 180,E1 -20512.7,E2 -20512.7} C_VEL
LIN {X 0,Y 221.504,Z 302.697,A -85,B 0,C 180,E1 -20518.182,E2 -20518.182} C_VEL
LIN {X 0,Y 221.504,Z 302.704,A -85,B 0,C 180,E1 -20521.818,E2 -20521.818} C_VEL
LIN {X 0,Y 221.252,Z 302.729,A -85,B 0,C 180,E1 -20527.299,E2 -20527.299} C_VEL
LIN {X 0,Y 221.061,Z 302.75,A -85,B 0,C 180,E1 -20530.997,E2 -20530.997} C_VEL
LIN {X 0,Y 221.008,Z 302.765,A -85,B 0,C 180,E1 -20536.63,E2 -20536.63} C_VEL
LIN {X 0,Y 220.878,Z 302.773,A -85,B 0,C 180,E1 -20540.487,E2 -20540.487} C_VEL
LIN {X 0,Y 220.856,Z 302.785,A -85,B 0,C 180,E1 -20544.436,E2 -20544.436} C_VEL
LIN {X 0,Y 220.821,Z 302.788,A -85,B 0,C 180,E1 -20548.515,E2 -20548.515} C_VEL
LIN {X 0,Y 220.811,Z 302.792,A -85,B 0,C 180,E1 -20552.757,E2 -20552.757} C_VEL
LIN {X 0,Y 220.805,Z 302.788,A -85,B 0,C 180,E1 -20557.279,E2 -20557.279} C_VEL
LIN {X 0,Y 220.766,Z 302.783,A -85,B 0,C 180,E1 -20561.953,E2 -20561.953} C_VEL
LIN {X 0,Y 220.772,Z 302.796,A -85,B 0,C 180,E1 -20565.547,E2 -20565.547} C_VEL
LIN {X 0,Y 220.804,Z 302.793,A -85,B 0,C 180,E1 -20570.464,E2 -20570.464} C_VEL
LIN {X 0,Y 220.802,Z 302.791,A -85,B 0,C 180,E1 -20573.043,E2 -20573.043} C_VEL
LIN {X 0,Y 220.038,Z 302.917,A -85,B 0,C 180,E1 -20574.086,E2 -20574.086} C_VEL
LIN {X 0,Y 214.406,Z 303.69,A -85,B 0,C 180,E1 -20577.358,E2 -20577.358} C_VEL
LIN {X 0,Y 213.984,Z 304.477,A -85,B 0,C 180,E1 -20578.185,E2 -20578.185} C_VEL
LIN {X 0,Y 214.027,Z 304.745,A -85,B 0,C 180,E1 -20578.342,E2 -20578.342} C_VEL
LIN {X 0,Y 215.552,Z 312.58,A -85,B 0,C 180,E1 -20582.314,E2 -20582.314} C_VEL
LIN {X 0,Y 215.78,Z 313.984,A -85,B 0,C 180,E1 -20583.005,E2 -20583.005} C_VEL
LIN {X 0,Y 218.648,Z 323.087,A -85,B 0,C 180,E1 -20583.668,E2 -20583.668} C_VEL
LIN {X 0,Y 223.002,Z 357.719,A -85,B 0,C 180,E1 -20585.358,E2 -20585.358} C_VEL
LIN {X 0,Y 222.868,Z 367,A -85,B 0,C 180,E1 -20585.679,E2 -20585.679} C_VEL
LIN {X 0,Y 222.004,Z 391.916,A -85,B 0,C 180,E1 -20586.563,E2 -20586.563} C_VEL
LIN {X 0,Y 221.22,Z 402.474,A -85,B 0,C 180,E1 -20587.19,E2 -20587.19} C_VEL
LIN {X 0,Y 220.103,Z 413.666,A -85,B 0,C 180,E1 -20588.218,E2 -20588.218} C_VEL
LIN {X 0,Y 218.977,Z 422.496,A -85,B 0,C 180,E1 -20589.327,E2 -20589.327} C_VEL
LIN {X 0,Y 217.618,Z 430.939,A -85,B 0,C 180,E1 -20590.67,E2 -20590.67} C_VEL
LIN {X 0,Y 216.541,Z 437.916,A -85,B 0,C 180,E1 -20592.042,E2 -20592.042} C_VEL
LIN {X 0,Y 215.535,Z 443.832,A -85,B 0,C 180,E1 -20593.423,E2 -20593.423} C_VEL
LIN {X 0,Y 214.328,Z 450.391,A -85,B 0,C 180,E1 -20595.278,E2 -20595.278} C_VEL
LIN {X 0,Y 213.39,Z 455.846,A -85,B 0,C 180,E1 -20597.156,E2 -20597.156} C_VEL
LIN {X 0,Y 212.501,Z 461.357,A -85,B 0,C 180,E1 -20599.52,E2 -20599.52} C_VEL
LIN {X 0,Y 211.993,Z 464.936,A -85,B 0,C 180,E1 -20601.421,E2 -20601.421} C_VEL
LIN {X 0,Y 211.565,Z 469.025,A -85,B 0,C 180,E1 -20604.281,E2 -20604.281} C_VEL
LIN {X 0,Y 211.44,Z 471.014,A -85,B 0,C 180,E1 -20606.188,E2 -20606.188} C_VEL
LIN {X 0,Y 211.468,Z 472.484,A -85,B 0,C 180,E1 -20608.095,E2 -20608.095} C_VEL
LIN {X 0,Y 211.56,Z 473.421,A -85,B 0,C 180,E1 -20610,E2 -20610} C_VEL
LIN {X 0,Y 211.448,Z 473.751,A -85,B 0,C 180,E1 -20611.905,E2 -20611.905} C_VEL
LIN {X 0,Y 211.418,Z 473.522,A -85,B 0,C 180,E1 -20614.241,E2 -20614.241} C_VEL
LIN {X 0,Y 211.84,Z 471.924,A -85,B 0,C 180,E1 -20617.626,E2 -20617.626} C_VEL
LIN {X 0,Y 212.659,Z 469.204,A -85,B 0,C 180,E1 -20620.472,E2 -20620.472} C_VEL
LIN {X 0,Y 213.436,Z 466.776,A -85,B 0,C 180,E1 -20622.358,E2 -20622.358} C_VEL
LIN {X 0,Y 215.06,Z 461.832,A -85,B 0,C 180,E1 -20625.155,E2 -20625.155} C_VEL
LIN {X 0,Y 216.814,Z 456.554,A -85,B 0,C 180,E1 -20627.447,E2 -20627.447} C_VEL
LIN {X 0,Y 218.426,Z 451.4,A -85,B 0,C 180,E1 -20629.256,E2 -20629.256} C_VEL
LIN {X 0,Y 220.325,Z 445.214,A -85,B 0,C 180,E1 -20631.029,E2 -20631.029} C_VEL
LIN {X 0,Y 222.194,Z 438.729,A -85,B 0,C 180,E1 -20632.551,E2 -20632.551} C_VEL
LIN {X 0,Y 223.884,Z 432.132,A -85,B 0,C 180,E1 -20633.838,E2 -20633.838} C_VEL
LIN {X 0,Y 225.669,Z 424.181,A -85,B 0,C 180,E1 -20635.107,E2 -20635.107} C_VEL
LIN {X 0,Y 227.244,Z 416.002,A -85,B 0,C 180,E1 -20636.149,E2 -20636.149} C_VEL
LIN {X 0,Y 228.837,Z 406.678,A -85,B 0,C 180,E1 -20637.046,E2 -20637.046} C_VEL
LIN {X 0,Y 230.267,Z 395.628,A -85,B 0,C 180,E1 -20637.804,E2 -20637.804} C_VEL
LIN {X 0,Y 231.192,Z 381.495,A -85,B 0,C 180,E1 -20638.368,E2 -20638.368} C_VEL
LIN {X 0,Y 231.922,Z 361.587,A -85,B 0,C 180,E1 -20639.036,E2 -20639.036} C_VEL
LIN {X 0,Y 230.147,Z 347.104,A -85,B 0,C 180,E1 -20639.925,E2 -20639.925} C_VEL
LIN {X 0,Y 228.417,Z 338.321,A -85,B 0,C 180,E1 -20640.6,E2 -20640.6} C_VEL
LIN {X 0,Y 222.368,Z 324.713,A -85,B 0,C 180,E1 -20642.361,E2 -20642.361} C_VEL
LIN {X 0,Y 217.7,Z 315.906,A -85,B 0,C 180,E1 -20643.746,E2 -20643.746} C_VEL
LIN {X 0,Y 215.946,Z 312.146,A -85,B 0,C 180,E1 -20644.373,E2 -20644.373} C_VEL
LIN {X 0,Y 214.153,Z 305.315,A -85,B 0,C 180,E1 -20648.573,E2 -20648.573} C_VEL
LIN {X 0,Y 213.764,Z 303.674,A -85,B 0,C 180,E1 -20649.72,E2 -20649.72} C_VEL
LIN {X 0,Y 213.699,Z 303.687,A -85,B 0,C 180,E1 -20653.679,E2 -20653.679} C_VEL
LIN {X 0,Y 213.699,Z 303.681,A -85,B 0,C 180,E1 -20656.344,E2 -20656.344} C_VEL
LIN {X 0,Y 213.712,Z 303.67,A -85,B 0,C 180,E1 -20659.143,E2 -20659.143} C_VEL
LIN {X 0,Y 213.739,Z 303.665,A -85,B 0,C 180,E1 -20663.711,E2 -20663.711} C_VEL
LIN {X 0,Y 213.763,Z 303.659,A -85,B 0,C 180,E1 -20668.262,E2 -20668.262} C_VEL
LIN {X 0,Y 213.821,Z 303.646,A -85,B 0,C 180,E1 -20672.603,E2 -20672.603} C_VEL
LIN {X 0,Y 213.813,Z 303.653,A -85,B 0,C 180,E1 -20676.974,E2 -20676.974} C_VEL
LIN {X 0,Y 213.937,Z 303.64,A -85,B 0,C 180,E1 -20682.803,E2 -20682.803} C_VEL
LIN {X 0,Y 213.945,Z 303.644,A -85,B 0,C 180,E1 -20686.706,E2 -20686.706} C_VEL
LIN {X 0,Y 214.135,Z 303.603,A -85,B 0,C 180,E1 -20690.555,E2 -20690.555} C_VEL
LIN {X 0,Y 214.201,Z 303.606,A -85,B 0,C 180,E1 -20692.459,E2 -20692.459} C_VEL
LIN {X 0,Y 214.436,Z 303.574,A -85,B 0,C 180,E1 -20698.122,E2 -20698.122} C_VEL
LIN {X 0,Y 214.542,Z 303.57,A -85,B 0,C 180,E1 -20700,E2 -20700} C_VEL
LIN {X 0,Y 214.435,Z 303.569,A -85,B 0,C 180,E1 -20701.878,E2 -20701.878} C_VEL
LIN {X 0,Y 214.175,Z 303.604,A -85,B 0,C 180,E1 -20707.542,E2 -20707.542} C_VEL
LIN {X 0,Y 213.992,Z 303.634,A -85,B 0,C 180,E1 -20711.365,E2 -20711.365} C_VEL
LIN {X 0,Y 213.924,Z 303.65,A -85,B 0,C 180,E1 -20715.238,E2 -20715.238} C_VEL
LIN {X 0,Y 213.834,Z 303.664,A -85,B 0,C 180,E1 -20719.188,E2 -20719.188} C_VEL
LIN {X 0,Y 213.843,Z 303.66,A -85,B 0,C 180,E1 -20723.228,E2 -20723.228} C_VEL
LIN {X 0,Y 213.831,Z 303.66,A -85,B 0,C 180,E1 -20727.207,E2 -20727.207} C_VEL
LIN {X 0,Y 214.785,Z 306.505,A -85,B 0,C 180,E1 -20727.595,E2 -20727.595} C_VEL
LIN {X 0,Y 216.609,Z 308.852,A -85,B 0,C 180,E1 -20728.13,E2 -20728.13} C_VEL
LIN {X 0,Y 219.717,Z 314.011,A -85,B 0,C 180,E1 -20729.065,E2 -20729.065} C_VEL
LIN {X 0,Y 225.003,Z 323.623,A -85,B 0,C 180,E1 -20730.575,E2 -20730.575} C_VEL
LIN {X 0,Y 231.044,Z 337.022,A -85,B 0,C 180,E1 -20732.281,E2 -20732.281} C_VEL
LIN {X 0,Y 232.854,Z 342.072,A -85,B 0,C 180,E1 -20732.799,E2 -20732.799} C_VEL
LIN {X 0,Y 230.894,Z 380.693,A -85,B 0,C 180,E1 -20734.073,E2 -20734.073} C_VEL
LIN {X 0,Y 229.873,Z 391.969,A -85,B 0,C 180,E1 -20734.722,E2 -20734.722} C_VEL
LIN {X 0,Y 228.329,Z 403.555,A -85,B 0,C 180,E1 -20735.791,E2 -20735.791} C_VEL
LIN {X 0,Y 226.92,Z 411.409,A -85,B 0,C 180,E1 -20736.74,E2 -20736.74} C_VEL
LIN {X 0,Y 225.169,Z 419.62,A -85,B 0,C 180,E1 -20737.994,E2 -20737.994} C_VEL
LIN {X 0,Y 223.25,Z 427.631,A -85,B 0,C 180,E1 -20739.534,E2 -20739.534} C_VEL
LIN {X 0,Y 221.528,Z 433.799,A -85,B 0,C 180,E1 -20740.974,E2 -20740.974} C_VEL
LIN {X 0,Y 219.709,Z 439.694,A -85,B 0,C 180,E1 -20742.634,E2 -20742.634} C_VEL
LIN {X 0,Y 218.191,Z 444.392,A -85,B 0,C 180,E1 -20744.221,E2 -20744.221} C_VEL
LIN {X 0,Y 216.665,Z 449.062,A -85,B 0,C 180,E1 -20746.145,E2 -20746.145} C_VEL
LIN {X 0,Y 214.858,Z 454.052,A -85,B 0,C 180,E1 -20748.793,E2 -20748.793} C_VEL
LIN {X 0,Y 213.545,Z 457.55,A -85,B 0,C 180,E1 -20751.296,E2 -20751.296} C_VEL
LIN {X 0,Y 212.617,Z 459.757,A -85,B 0,C 180,E1 -20753.49,E2 -20753.49} C_VEL
LIN {X 0,Y 211.923,Z 461.392,A -85,B 0,C 180,E1 -20756.004,E2 -20756.004} C_VEL
LIN {X 0,Y 211.52,Z 462.042,A -85,B 0,C 180,E1 -20757.886,E2 -20757.886} C_VEL
LIN {X 0,Y 211.239,Z 462.192,A -85,B 0,C 180,E1 -20760.064,E2 -20760.064} C_VEL
LIN {X 0,Y 211.109,Z 461.71,A -85,B 0,C 180,E1 -20762.221,E2 -20762.221} C_VEL
LIN {X 0,Y 211.21,Z 460.566,A -85,B 0,C 180,E1 -20764.37,E2 -20764.37} C_VEL
LIN {X 0,Y 211.742,Z 457.644,A -85,B 0,C 180,E1 -20767.473,E2 -20767.473} C_VEL
LIN {X 0,Y 212.148,Z 454.746,A -85,B 0,C 180,E1 -20769.645,E2 -20769.645} C_VEL
LIN {X 0,Y 212.939,Z 450.16,A -85,B 0,C 180,E1 -20772.225,E2 -20772.225} C_VEL
LIN {X 0,Y 213.945,Z 444.305,A -85,B 0,C 180,E1 -20774.764,E2 -20774.764} C_VEL
LIN {X 0,Y 215.411,Z 436.396,A -85,B 0,C 180,E1 -20777.409,E2 -20777.409} C_VEL
LIN {X 0,Y 216.818,Z 428.199,A -85,B 0,C 180,E1 -20779.495,E2 -20779.495} C_VEL
LIN {X 0,Y 217.949,Z 421.153,A -85,B 0,C 180,E1 -20780.956,E2 -20780.956} C_VEL
LIN {X 0,Y 219.248,Z 412.5,A -85,B 0,C 180,E1 -20782.402,E2 -20782.402} C_VEL
LIN {X 0,Y 220.334,Z 403.501,A -85,B 0,C 180,E1 -20783.59,E2 -20783.59} C_VEL
LIN {X 0,Y 221.393,Z 392.286,A -85,B 0,C 180,E1 -20784.704,E2 -20784.704} C_VEL
LIN {X 0,Y 222.174,Z 381.441,A -85,B 0,C 180,E1 -20785.396,E2 -20785.396} C_VEL
LIN {X 0,Y 222.998,Z 358.953,A -85,B 0,C 180,E1 -20786.21,E2 -20786.21} C_VEL
LIN {X 0,Y 223.598,Z 335.915,A -85,B 0,C 180,E1 -20786.985,E2 -20786.985} C_VEL
LIN {X 0,Y 221.679,Z 325.082,A -85,B 0,C 180,E1 -20787.564,E2 -20787.564} C_VEL
LIN {X 0,Y 215.019,Z 305.487,A -85,B 0,C 180,E1 -20788.983,E2 -20788.983} C_VEL
LIN {X 0,Y 214.482,Z 303.585,A -85,B 0,C 180,E1 -20789.121,E2 -20789.121} C_VEL
LIN {X 0,Y 214.446,Z 303.587,A -85,B 0,C 180,E1 -20791.878,E2 -20791.878} C_VEL
LIN {X 0,Y 214.191,Z 303.615,A -85,B 0,C 180,E1 -20797.541,E2 -20797.541} C_VEL
LIN {X 0,Y 213.999,Z 303.634,A -85,B 0,C 180,E1 -20801.364,E2 -20801.364} C_VEL
LIN {X 0,Y 213.914,Z 303.65,A -85,B 0,C 180,E1 -20805.238,E2 -20805.238} C_VEL
LIN {X 0,Y 213.817,Z 303.655,A -85,B 0,C 180,E1 -20809.189,E2 -20809.189} C_VEL
LIN {X 0,Y 213.811,Z 303.653,A -85,B 0,C 180,E1 -20813.23,E2 -20813.23} C_VEL
LIN {X 0,Y 213.829,Z 303.664,A -85,B 0,C 180,E1 -20817.449,E2 -20817.449} C_VEL
LIN {X 0,Y 213.777,Z 303.663,A -85,B 0,C 180,E1 -20821.735,E2 -20821.735} C_VEL
LIN {X 0,Y 213.742,Z 303.672,A -85,B 0,C 180,E1 -20826.287,E2 -20826.287} C_VEL
LIN {X 0,Y 213.713,Z 303.67,A -85,B 0,C 180,E1 -20831.124,E2 -20831.124} C_VEL
LIN {X 0,Y 213.807,Z 303.662,A -85,B 0,C 180,E1 -20836.314,E2 -20836.314} C_VEL
LIN {X 0,Y 213.792,Z 303.665,A -85,B 0,C 180,E1 -20839.118,E2 -20839.118} C_VEL
LIN {X 0,Y 213.751,Z 303.659,A -85,B 0,C 180,E1 -20843.713,E2 -20843.713} C_VEL
LIN {X 0,Y 213.792,Z 303.662,A -85,B 0,C 180,E1 -20848.724,E2 -20848.724} C_VEL
LIN {X 0,Y 213.822,Z 303.661,A -85,B 0,C 180,E1 -20852.602,E2 -20852.602} C_VEL
LIN {X 0,Y 213.847,Z 303.647,A -85,B 0,C 180,E1 -20856.952,E2 -20856.952} C_VEL
LIN {X 0,Y 213.938,Z 303.643,A -85,B 0,C 180,E1 -20862.803,E2 -20862.803} C_VEL
LIN {X 0,Y 213.946,Z 303.649,A -85,B 0,C 180,E1 -20866.706,E2 -20866.706} C_VEL
LIN {X 0,Y 214.136,Z 303.621,A -85,B 0,C 180,E1 -20870.555,E2 -20870.555} C_VEL
LIN {X 0,Y 214.092,Z 303.613,A -85,B 0,C 180,E1 -20874.348,E2 -20874.348} C_VEL
LIN {X 0,Y 214.437,Z 303.577,A -85,B 0,C 180,E1 -20878.122,E2 -20878.122} C_VEL
LIN {X 0,Y 214.543,Z 303.569,A -85,B 0,C 180,E1 -20880,E2 -20880} C_VEL
LIN {X 0,Y 214.437,Z 303.584,A -85,B 0,C 180,E1 -20881.878,E2 -20881.878} C_VEL
LIN {X 0,Y 214.191,Z 303.606,A -85,B 0,C 180,E1 -20887.541,E2 -20887.541} C_VEL
LIN {X 0,Y 213.993,Z 303.632,A -85,B 0,C 180,E1 -20891.364,E2 -20891.364} C_VEL
LIN {X 0,Y 213.924,Z 303.649,A -85,B 0,C 180,E1 -20895.237,E2 -20895.237} C_VEL
LIN {X 0,Y 213.829,Z 303.657,A -85,B 0,C 180,E1 -20899.188,E2 -20899.188} C_VEL
LIN {X 0,Y 213.805,Z 303.658,A -85,B 0,C 180,E1 -20903.232,E2 -20903.232} C_VEL
LIN {X 0,Y 213.824,Z 303.661,A -85,B 0,C 180,E1 -20907.45,E2 -20907.45} C_VEL
LIN {X 0,Y 213.763,Z 303.665,A -85,B 0,C 180,E1 -20911.738,E2 -20911.738} C_VEL
LIN {X 0,Y 213.739,Z 303.674,A -85,B 0,C 180,E1 -20916.289,E2 -20916.289} C_VEL
LIN {X 0,Y 213.708,Z 303.66,A -85,B 0,C 180,E1 -20921.126,E2 -20921.126} C_VEL
LIN {X 0,Y 213.703,Z 303.672,A -85,B 0,C 180,E1 -20923.679,E2 -20923.679} C_VEL
LIN {X 0,Y 213.704,Z 303.677,A -85,B 0,C 180,E1 -20926.344,E2 -20926.344} C_VEL
LIN {X 0,Y 213.714,Z 303.677,A -85,B 0,C 180,E1 -20929.144,E2 -20929.144} C_VEL
LIN {X 0,Y 213.741,Z 303.672,A -85,B 0,C 180,E1 -20933.712,E2 -20933.712} C_VEL
LIN {X 0,Y 213.837,Z 303.818,A -85,B 0,C 180,E1 -20937.859,E2 -20937.859} C_VEL
LIN {X 0,Y 214.027,Z 304.745,A -85,B 0,C 180,E1 -20938.342,E2 -20938.342} C_VEL
LIN {X 0,Y 213.76,Z 306.849,A -85,B 0,C 180,E1 -20939.343,E2 -20939.343} C_VEL
LIN {X 0,Y 211.306,Z 310.884,A -85,B 0,C 180,E1 -20941.033,E2 -20941.033} C_VEL
LIN {X 0,Y 209.867,Z 314.565,A -85,B 0,C 180,E1 -20942.027,E2 -20942.027} C_VEL
LIN {X 0,Y 209.835,Z 317.649,A -85,B 0,C 180,E1 -20942.512,E2 -20942.512} C_VEL
LIN {X 0,Y 210.053,Z 318.546,A -85,B 0,C 180,E1 -20942.593,E2 -20942.593} C_VEL
LIN {X 0,Y 212.161,Z 325.095,A -85,B 0,C 180,E1 -20943.072,E2 -20943.072} C_VEL
LIN {X 0,Y 216.268,Z 357.881,A -85,B 0,C 180,E1 -20944.733,E2 -20944.733} C_VEL
LIN {X 0,Y 216.224,Z 365.3,A -85,B 0,C 180,E1 -20945.006,E2 -20945.006} C_VEL
LIN {X 0,Y 215.268,Z 392.751,A -85,B 0,C 180,E1 -20946.018,E2 -20946.018} C_VEL
LIN {X 0,Y 214.156,Z 404.826,A -85,B 0,C 180,E1 -20946.809,E2 -20946.809} C_VEL
LIN {X 0,Y 213.157,Z 414.87,A -85,B 0,C 180,E1 -20947.843,E2 -20947.843} C_VEL
LIN {X 0,Y 212.098,Z 422.732,A -85,B 0,C 180,E1 -20948.879,E2 -20948.879} C_VEL
LIN {X 0,Y 210.689,Z 431.098,A -85,B 0,C 180,E1 -20950.261,E2 -20950.261} C_VEL
LIN {X 0,Y 209.587,Z 438.016,A -85,B 0,C 180,E1 -20951.678,E2 -20951.678} C_VEL
LIN {X 0,Y 208.366,Z 444.742,A -85,B 0,C 180,E1 -20953.34,E2 -20953.34} C_VEL
LIN {X 0,Y 207.173,Z 451.121,A -85,B 0,C 180,E1 -20955.261,E2 -20955.261} C_VEL
LIN {X 0,Y 206.232,Z 456.415,A -85,B 0,C 180,E1 -20957.203,E2 -20957.203} C_VEL
LIN {X 0,Y 205.502,Z 460.819,A -85,B 0,C 180,E1 -20959.159,E2 -20959.159} C_VEL
LIN {X 0,Y 204.761,Z 466.003,A -85,B 0,C 180,E1 -20962.109,E2 -20962.109} C_VEL
LIN {X 0,Y 204.495,Z 468.623,A -85,B 0,C 180,E1 -20964.082,E2 -20964.082} C_VEL
LIN {X 0,Y 204.364,Z 470.675,A -85,B 0,C 180,E1 -20966.056,E2 -20966.056} C_VEL
LIN {X 0,Y 204.371,Z 472.201,A -85,B 0,C 180,E1 -20968.029,E2 -20968.029} C_VEL
LIN {X 0,Y 204.477,Z 473.152,A -85,B 0,C 180,E1 -20970,E2 -20970} C_VEL
LIN {X 0,Y 204.352,Z 473.525,A -85,B 0,C 180,E1 -20971.971,E2 -20971.971} C_VEL
LIN {X 0,Y 204.326,Z 473.411,A -85,B 0,C 180,E1 -20974.066,E2 -20974.066} C_VEL
LIN {X 0,Y 204.497,Z 472.884,A -85,B 0,C 180,E1 -20975.918,E2 -20975.918} C_VEL
LIN {X 0,Y 204.783,Z 471.848,A -85,B 0,C 180,E1 -20977.89,E2 -20977.89} C_VEL
LIN {X 0,Y 205.685,Z 469.214,A -85,B 0,C 180,E1 -20980.832,E2 -20980.832} C_VEL
LIN {X 0,Y 206.492,Z 466.84,A -85,B 0,C 180,E1 -20982.781,E2 -20982.781} C_VEL
LIN {X 0,Y 208.205,Z 462.004,A -85,B 0,C 180,E1 -20985.666,E2 -20985.666} C_VEL
LIN {X 0,Y 210.07,Z 456.808,A -85,B 0,C 180,E1 -20988.026,E2 -20988.026} C_VEL
LIN {X 0,Y 211.755,Z 451.746,A -85,B 0,C 180,E1 -20989.888,E2 -20989.888} C_VEL
LIN {X 0,Y 213.743,Z 445.666,A -85,B 0,C 180,E1 -20991.709,E2 -20991.709} C_VEL
LIN {X 0,Y 215.99,Z 438.29,A -85,B 0,C 180,E1 -20993.49,E2 -20993.49} C_VEL
LIN {X 0,Y 217.783,Z 431.642,A -85,B 0,C 180,E1 -20994.803,E2 -20994.803} C_VEL
LIN {X 0,Y 219.575,Z 423.684,A -85,B 0,C 180,E1 -20996.102,E2 -20996.102} C_VEL
LIN {X 0,Y 221.309,Z 415.363,A -85,B 0,C 180,E1 -20997.161,E2 -20997.161} C_VEL
LIN {X 0,Y 222.791,Z 406.986,A -85,B 0,C 180,E1 -20997.984,E2 -20997.984} C_VEL
LIN {X 0,Y 224.131,Z 397.294,A -85,B 0,C 180,E1 -20998.682,E2 -20998.682} C_VEL
LIN {X 0,Y 225.074,Z 386.069,A -85,B 0,C 180,E1 -20999.222,E2 -20999.222} C_VEL
LIN {X 0,Y 226.041,Z 362.387,A -85,B 0,C 180,E1 -21000.035,E2 -21000.035} C_VEL
LIN {X 0,Y 224.387,Z 348.469,A -85,B 0,C 180,E1 -21000.933,E2 -21000.933} C_VEL
LIN {X 0,Y 223.022,Z 341.302,A -85,B 0,C 180,E1 -21001.507,E2 -21001.507} C_VEL
LIN {X 0,Y 217.448,Z 328.667,A -85,B 0,C 180,E1 -21003.216,E2 -21003.216} C_VEL
LIN {X 0,Y 211.22,Z 316.65,A -85,B 0,C 180,E1 -21005.227,E2 -21005.227} C_VEL
LIN {X 0,Y 208.942,Z 312.637,A -85,B 0,C 180,E1 -21005.998,E2 -21005.998} C_VEL
LIN {X 0,Y 208.633,Z 311.852,A -85,B 0,C 180,E1 -21006.175,E2 -21006.175} C_VEL
LIN {X 0,Y 206.972,Z 305.797,A -85,B 0,C 180,E1 -21010.177,E2 -21010.177} C_VEL
LIN {X 0,Y 206.67,Z 304.561,A -85,B 0,C 180,E1 -21011.049,E2 -21011.049} C_VEL
LIN {X 0,Y 206.627,Z 304.558,A -85,B 0,C 180,E1 -21015.582,E2 -21015.582} C_VEL
LIN {X 0,Y 206.656,Z 304.551,A -85,B 0,C 180,E1 -21019.748,E2 -21019.748} C_VEL
LIN {X 0,Y 206.695,Z 304.551,A -85,B 0,C 180,E1 -21024.688,E2 -21024.688} C_VEL
LIN {X 0,Y 206.71,Z 304.546,A -85,B 0,C 180,E1 -21029.337,E2 -21029.337} C_VEL
LIN {X 0,Y 206.725,Z 304.534,A -85,B 0,C 180,E1 -21033.771,E2 -21033.771} C_VEL
LIN {X 0,Y 206.732,Z 304.527,A -85,B 0,C 180,E1 -21038.041,E2 -21038.041} C_VEL
LIN {X 0,Y 206.867,Z 304.525,A -85,B 0,C 180,E1 -21042.196,E2 -21042.196} C_VEL
LIN {X 0,Y 206.888,Z 304.519,A -85,B 0,C 180,E1 -21046.244,E2 -21046.244} C_VEL
LIN {X 0,Y 207.094,Z 304.481,A -85,B 0,C 180,E1 -21050.231,E2 -21050.231} C_VEL
LIN {X 0,Y 207.056,Z 304.503,A -85,B 0,C 180,E1 -21054.156,E2 -21054.156} C_VEL
LIN {X 0,Y 207.373,Z 304.452,A -85,B 0,C 180,E1 -21058.058,E2 -21058.058} C_VEL
LIN {X 0,Y 207.507,Z 304.446,A -85,B 0,C 180,E1 -21060,E2 -21060} C_VEL
LIN {X 0,Y 207.371,Z 304.448,A -85,B 0,C 180,E1 -21061.942,E2 -21061.942} C_VEL
LIN {X 0,Y 207.119,Z 304.483,A -85,B 0,C 180,E1 -21067.801,E2 -21067.801} C_VEL
LIN {X 0,Y 206.917,Z 304.513,A -85,B 0,C 180,E1 -21071.759,E2 -21071.759} C_VEL
LIN {X 0,Y 206.858,Z 304.526,A -85,B 0,C 180,E1 -21075.772,E2 -21075.772} C_VEL
LIN {X 0,Y 206.778,Z 304.538,A -85,B 0,C 180,E1 -21079.87,E2 -21079.87} C_VEL
LIN {X 0,Y 206.759,Z 304.541,A -85,B 0,C 180,E1 -21084.073,E2 -21084.073} C_VEL
LIN {X 0,Y 206.764,Z 304.562,A -85,B 0,C 180,E1 -21085.48,E2 -21085.48} C_VEL
LIN {X 0,Y 207.76,Z 307.324,A -85,B 0,C 180,E1 -21085.886,E2 -21085.886} C_VEL
LIN {X 0,Y 209.718,Z 309.737,A -85,B 0,C 180,E1 -21086.514,E2 -21086.514} C_VEL
LIN {X 0,Y 211.768,Z 313.041,A -85,B 0,C 180,E1 -21087.186,E2 -21087.186} C_VEL
LIN {X 0,Y 215.242,Z 318.619,A -85,B 0,C 180,E1 -21088.275,E2 -21088.275} C_VEL
LIN {X 0,Y 220.441,Z 328.422,A -85,B 0,C 180,E1 -21089.861,E2 -21089.861} C_VEL
LIN {X 0,Y 225.849,Z 340.603,A -85,B 0,C 180,E1 -21091.465,E2 -21091.465} C_VEL
LIN {X 0,Y 227.001,Z 343.635,A -85,B 0,C 180,E1 -21091.81,E2 -21091.81} C_VEL
LIN {X 0,Y 225.014,Z 381.022,A -85,B 0,C 180,E1 -21093.08,E2 -21093.08} C_VEL
LIN {X 0,Y 223.943,Z 392.161,A -85,B 0,C 180,E1 -21093.736,E2 -21093.736} C_VEL
LIN {X 0,Y 222.426,Z 403.194,A -85,B 0,C 180,E1 -21094.765,E2 -21094.765} C_VEL
LIN {X 0,Y 220.886,Z 411.436,A -85,B 0,C 180,E1 -21095.775,E2 -21095.775} C_VEL
LIN {X 0,Y 219.016,Z 419.805,A -85,B 0,C 180,E1 -21097.077,E2 -21097.077} C_VEL
LIN {X 0,Y 217.181,Z 427.103,A -85,B 0,C 180,E1 -21098.493,E2 -21098.493} C_VEL
LIN {X 0,Y 215.395,Z 433.29,A -85,B 0,C 180,E1 -21099.938,E2 -21099.938} C_VEL
LIN {X 0,Y 213.568,Z 439.017,A -85,B 0,C 180,E1 -21101.544,E2 -21101.544} C_VEL
LIN {X 0,Y 211.243,Z 445.65,A -85,B 0,C 180,E1 -21103.877,E2 -21103.877} C_VEL
LIN {X 0,Y 209.643,Z 450.248,A -85,B 0,C 180,E1 -21105.926,E2 -21105.926} C_VEL
LIN {X 0,Y 208.206,Z 453.936,A -85,B 0,C 180,E1 -21107.955,E2 -21107.955} C_VEL
LIN {X 0,Y 206.651,Z 457.837,A -85,B 0,C 180,E1 -21110.817,E2 -21110.817} C_VEL
LIN {X 0,Y 206.005,Z 459.233,A -85,B 0,C 180,E1 -21112.116,E2 -21112.116} C_VEL
LIN {X 0,Y 205.222,Z 461.013,A -85,B 0,C 180,E1 -21114.397,E2 -21114.397} C_VEL
LIN {X 0,Y 204.657,Z 462.076,A -85,B 0,C 180,E1 -21116.672,E2 -21116.672} C_VEL
LIN {X 0,Y 204.205,Z 462.463,A -85,B 0,C 180,E1 -21119.363,E2 -21119.363} C_VEL
LIN {X 0,Y 204.038,Z 462.153,A -85,B 0,C 180,E1 -21121.17,E2 -21121.17} C_VEL
LIN {X 0,Y 204.058,Z 461.146,A -85,B 0,C 180,E1 -21123.57,E2 -21123.57} C_VEL
LIN {X 0,Y 204.468,Z 458.728,A -85,B 0,C 180,E1 -21126.717,E2 -21126.717} C_VEL
LIN {X 0,Y 204.927,Z 456.076,A -85,B 0,C 180,E1 -21128.967,E2 -21128.967} C_VEL
LIN {X 0,Y 205.782,Z 450.96,A -85,B 0,C 180,E1 -21132.1,E2 -21132.1} C_VEL
LIN {X 0,Y 206.533,Z 446.524,A -85,B 0,C 180,E1 -21134.204,E2 -21134.204} C_VEL
LIN {X 0,Y 207.589,Z 441.083,A -85,B 0,C 180,E1 -21136.292,E2 -21136.292} C_VEL
LIN {X 0,Y 208.812,Z 434.468,A -85,B 0,C 180,E1 -21138.35,E2 -21138.35} C_VEL
LIN {X 0,Y 210.05,Z 427.461,A -85,B 0,C 180,E1 -21140.127,E2 -21140.127} C_VEL
LIN {X 0,Y 211.274,Z 420.208,A -85,B 0,C 180,E1 -21141.632,E2 -21141.632} C_VEL
LIN {X 0,Y 212.448,Z 412.443,A -85,B 0,C 180,E1 -21142.947,E2 -21142.947} C_VEL
LIN {X 0,Y 213.566,Z 403.614,A -85,B 0,C 180,E1 -21144.141,E2 -21144.141} C_VEL
LIN {X 0,Y 214.686,Z 392.136,A -85,B 0,C 180,E1 -21145.306,E2 -21145.306} C_VEL
LIN {X 0,Y 215.506,Z 380.803,A -85,B 0,C 180,E1 -21146.026,E2 -21146.026} C_VEL
LIN {X 0,Y 216.659,Z 349.808,A -85,B 0,C 180,E1 -21147.142,E2 -21147.142} C_VEL
LIN {X 0,Y 216.89,Z 336.646,A -85,B 0,C 180,E1 -21147.612,E2 -21147.612} C_VEL
LIN {X 0,Y 215.292,Z 327.234,A -85,B 0,C 180,E1 -21148.129,E2 -21148.129} C_VEL
LIN {X 0,Y 208.923,Z 308.535,A -85,B 0,C 180,E1 -21149.54,E2 -21149.54} C_VEL
LIN {X 0,Y 207.498,Z 304.455,A -85,B 0,C 180,E1 -21149.879,E2 -21149.879} C_VEL
LIN {X 0,Y 207.382,Z 304.466,A -85,B 0,C 180,E1 -21151.942,E2 -21151.942} C_VEL
LIN {X 0,Y 207.134,Z 304.495,A -85,B 0,C 180,E1 -21157.8,E2 -21157.8} C_VEL
LIN {X 0,Y 206.922,Z 304.513,A -85,B 0,C 180,E1 -21161.758,E2 -21161.758} C_VEL
LIN {X 0,Y 206.847,Z 304.53,A -85,B 0,C 180,E1 -21165.772,E2 -21165.772} C_VEL
LIN {X 0,Y 206.858,Z 304.528,A -85,B 0,C 180,E1 -21167.954,E2 -21167.954} C_VEL
LIN {X 0,Y 206.754,Z 304.533,A -85,B 0,C 180,E1 -21173.395,E2 -21173.395} C_VEL
LIN {X 0,Y 206.744,Z 304.547,A -85,B 0,C 180,E1 -21178.418,E2 -21178.418} C_VEL
LIN {X 0,Y 206.702,Z 304.544,A -85,B 0,C 180,E1 -21182.956,E2 -21182.956} C_VEL
LIN {X 0,Y 206.679,Z 304.553,A -85,B 0,C 180,E1 -21187.739,E2 -21187.739} C_VEL
LIN {X 0,Y 206.645,Z 304.546,A -85,B 0,C 180,E1 -21191.563,E2 -21191.563} C_VEL
LIN {X 0,Y 206.702,Z 304.547,A -85,B 0,C 180,E1 -21195.56,E2 -21195.56} C_VEL
LIN {X 0,Y 206.722,Z 304.546,A -85,B 0,C 180,E1 -21199.763,E2 -21199.763} C_VEL
LIN {X 0,Y 206.722,Z 304.538,A -85,B 0,C 180,E1 -21202.269,E2 -21202.269} C_VEL
LIN {X 0,Y 206.706,Z 304.539,A -85,B 0,C 180,E1 -21207.043,E2 -21207.043} C_VEL
LIN {X 0,Y 206.763,Z 304.543,A -85,B 0,C 180,E1 -21212.096,E2 -21212.096} C_VEL
LIN {X 0,Y 206.781,Z 304.529,A -85,B 0,C 180,E1 -21216.583,E2 -21216.583} C_VEL
LIN {X 0,Y 206.868,Z 304.518,A -85,B 0,C 180,E1 -21222.196,E2 -21222.196} C_VEL
LIN {X 0,Y 206.888,Z 304.525,A -85,B 0,C 180,E1 -21226.244,E2 -21226.244} C_VEL
LIN {X 0,Y 207.094,Z 304.497,A -85,B 0,C 180,E1 -21230.23,E2 -21230.23} C_VEL
LIN {X 0,Y 207.053,Z 304.489,A -85,B 0,C 180,E1 -21234.155,E2 -21234.155} C_VEL
LIN {X 0,Y 207.374,Z 304.456,A -85,B 0,C 180,E1 -21238.058,E2 -21238.058} C_VEL
LIN {X 0,Y 207.508,Z 304.445,A -85,B 0,C 180,E1 -21240,E2 -21240} C_VEL
LIN {X 0,Y 207.374,Z 304.464,A -85,B 0,C 180,E1 -21241.942,E2 -21241.942} C_VEL
LIN {X 0,Y 207.134,Z 304.483,A -85,B 0,C 180,E1 -21247.8,E2 -21247.8} C_VEL
LIN {X 0,Y 206.918,Z 304.516,A -85,B 0,C 180,E1 -21251.758,E2 -21251.758} C_VEL
LIN {X 0,Y 206.858,Z 304.531,A -85,B 0,C 180,E1 -21255.771,E2 -21255.771} C_VEL
LIN {X 0,Y 206.756,Z 304.535,A -85,B 0,C 180,E1 -21259.872,E2 -21259.872} C_VEL
LIN {X 0,Y 206.742,Z 304.543,A -85,B 0,C 180,E1 -21264.075,E2 -21264.075} C_VEL
LIN {X 0,Y 206.732,Z 304.543,A -85,B 0,C 180,E1 -21268.42,E2 -21268.42} C_VEL
LIN {X 0,Y 206.694,Z 304.55,A -85,B 0,C 180,E1 -21272.958,E2 -21272.958} C_VEL
LIN {X 0,Y 206.675,Z 304.549,A -85,B 0,C 180,E1 -21277.741,E2 -21277.741} C_VEL
LIN {X 0,Y 206.638,Z 304.541,A -85,B 0,C 180,E1 -21281.563,E2 -21281.563} C_VEL
LIN {X 0,Y 206.631,Z 304.557,A -85,B 0,C 180,E1 -21285.582,E2 -21285.582} C_VEL
LIN {X 0,Y 206.658,Z 304.554,A -85,B 0,C 180,E1 -21289.75,E2 -21289.75} C_VEL
LIN {X 0,Y 206.697,Z 304.551,A -85,B 0,C 180,E1 -21294.689,E2 -21294.689} C_VEL
LIN {X 0,Y 206.777,Z 304.581,A -85,B 0,C 180,E1 -21297.364,E2 -21297.364} C_VEL
LIN {X 0,Y 208.482,Z 313.049,A -85,B 0,C 180,E1 -21301.84,E2 -21301.84} C_VEL
LIN {X 0,Y 208.615,Z 313.96,A -85,B 0,C 180,E1 -21302.255,E2 -21302.255} C_VEL
LIN {X 0,Y 210.053,Z 318.546,A -85,B 0,C 180,E1 -21302.593,E2 -21302.593} C_VEL
LIN {X 0,Y 210.806,Z 322.31,A -85,B 0,C 180,E1 -21302.82,E2 -21302.82} C_VEL
LIN {X 0,Y 210.931,Z 326.204,A -85,B 0,C 180,E1 -21302.983,E2 -21302.983} C_VEL
LIN {X 0,Y 210.036,Z 334.092,A -85,B 0,C 180,E1 -21303.192,E2 -21303.192} C_VEL
LIN {X 0,Y 208.574,Z 344.036,A -85,B 0,C 180,E1 -21303.423,E2 -21303.423} C_VEL
LIN {X 0,Y 208.645,Z 349.977,A -85,B 0,C 180,E1 -21303.663,E2 -21303.663} C_VEL
LIN {X 0,Y 209.753,Z 361.784,A -85,B 0,C 180,E1 -21304.234,E2 -21304.234} C_VEL
LIN {X 0,Y 208.615,Z 391.094,A -85,B 0,C 180,E1 -21305.315,E2 -21305.315} C_VEL
LIN {X 0,Y 207.849,Z 401.116,A -85,B 0,C 180,E1 -21305.931,E2 -21305.931} C_VEL
LIN {X 0,Y 206.774,Z 411.116,A -85,B 0,C 180,E1 -21306.836,E2 -21306.836} C_VEL
LIN {X 0,Y 205.502,Z 421.471,A -85,B 0,C 180,E1 -21308.167,E2 -21308.167} C_VEL
LIN {X 0,Y 204.002,Z 430.022,A -85,B 0,C 180,E1 -21309.586,E2 -21309.586} C_VEL
LIN {X 0,Y 202.642,Z 438.117,A -85,B 0,C 180,E1 -21311.289,E2 -21311.289} C_VEL
LIN {X 0,Y 201.571,Z 443.937,A -85,B 0,C 180,E1 -21312.761,E2 -21312.761} C_VEL
LIN {X 0,Y 200.285,Z 450.413,A -85,B 0,C 180,E1 -21314.742,E2 -21314.742} C_VEL
LIN {X 0,Y 199.285,Z 455.796,A -85,B 0,C 180,E1 -21316.749,E2 -21316.749} C_VEL
LIN {X 0,Y 198.497,Z 460.277,A -85,B 0,C 180,E1 -21318.771,E2 -21318.771} C_VEL
LIN {X 0,Y 197.714,Z 465.531,A -85,B 0,C 180,E1 -21321.826,E2 -21321.826} C_VEL
LIN {X 0,Y 197.412,Z 468.217,A -85,B 0,C 180,E1 -21323.869,E2 -21323.869} C_VEL
LIN {X 0,Y 197.285,Z 470.331,A -85,B 0,C 180,E1 -21325.914,E2 -21325.914} C_VEL
LIN {X 0,Y 197.277,Z 471.904,A -85,B 0,C 180,E1 -21327.958,E2 -21327.958} C_VEL
LIN {X 0,Y 197.396,Z 472.867,A -85,B 0,C 180,E1 -21330,E2 -21330} C_VEL
LIN {X 0,Y 197.258,Z 473.296,A -85,B 0,C 180,E1 -21332.042,E2 -21332.042} C_VEL
LIN {X 0,Y 197.246,Z 473.266,A -85,B 0,C 180,E1 -21334.086,E2 -21334.086} C_VEL
LIN {X 0,Y 197.415,Z 472.78,A -85,B 0,C 180,E1 -21336.131,E2 -21336.131} C_VEL
LIN {X 0,Y 197.738,Z 471.768,A -85,B 0,C 180,E1 -21338.173,E2 -21338.173} C_VEL
LIN {X 0,Y 198.697,Z 469.241,A -85,B 0,C 180,E1 -21341.217,E2 -21341.217} C_VEL
LIN {X 0,Y 200.1,Z 465.425,A -85,B 0,C 180,E1 -21344.232,E2 -21344.232} C_VEL
LIN {X 0,Y 202.104,Z 460.247,A -85,B 0,C 180,E1 -21347.192,E2 -21347.192} C_VEL
LIN {X 0,Y 204.175,Z 454.704,A -85,B 0,C 180,E1 -21349.609,E2 -21349.609} C_VEL
LIN {X 0,Y 206.626,Z 447.793,A -85,B 0,C 180,E1 -21351.971,E2 -21351.971} C_VEL
LIN {X 0,Y 209.54,Z 438.896,A -85,B 0,C 180,E1 -21354.258,E2 -21354.258} C_VEL
LIN {X 0,Y 211.389,Z 432.433,A -85,B 0,C 180,E1 -21355.607,E2 -21355.607} C_VEL
LIN {X 0,Y 213.251,Z 424.938,A -85,B 0,C 180,E1 -21356.895,E2 -21356.895} C_VEL
LIN {X 0,Y 215.06,Z 416.713,A -85,B 0,C 180,E1 -21358.019,E2 -21358.019} C_VEL
LIN {X 0,Y 216.8,Z 407.614,A -85,B 0,C 180,E1 -21358.961,E2 -21358.961} C_VEL
LIN {X 0,Y 218.166,Z 398.529,A -85,B 0,C 180,E1 -21359.652,E2 -21359.652} C_VEL
LIN {X 0,Y 219.095,Z 388.79,A -85,B 0,C 180,E1 -21360.171,E2 -21360.171} C_VEL
LIN {X 0,Y 220.305,Z 363.194,A -85,B 0,C 180,E1 -21361.09,E2 -21361.09} C_VEL
LIN {X 0,Y 218.62,Z 349.17,A -85,B 0,C 180,E1 -21362.046,E2 -21362.046} C_VEL
LIN {X 0,Y 217.58,Z 344.024,A -85,B 0,C 180,E1 -21362.492,E2 -21362.492} C_VEL
LIN {X 0,Y 212.165,Z 331.727,A -85,B 0,C 180,E1 -21364.271,E2 -21364.271} C_VEL
LIN {X 0,Y 206.715,Z 321.155,A -85,B 0,C 180,E1 -21366.133,E2 -21366.133} C_VEL
LIN {X 0,Y 203.602,Z 315.876,A -85,B 0,C 180,E1 -21367.239,E2 -21367.239} C_VEL
LIN {X 0,Y 201.477,Z 312.082,A -85,B 0,C 180,E1 -21368.04,E2 -21368.04} C_VEL
LIN {X 0,Y 201.288,Z 311.574,A -85,B 0,C 180,E1 -21368.167,E2 -21368.167} C_VEL
LIN {X 0,Y 199.574,Z 305.441,A -85,B 0,C 180,E1 -21372.629,E2 -21372.629} C_VEL
LIN {X 0,Y 199.568,Z 305.437,A -85,B 0,C 180,E1 -21377.69,E2 -21377.69} C_VEL
LIN {X 0,Y 199.607,Z 305.435,A -85,B 0,C 180,E1 -21380.767,E2 -21380.767} C_VEL
LIN {X 0,Y 199.608,Z 305.43,A -85,B 0,C 180,E1 -21385.713,E2 -21385.713} C_VEL
LIN {X 0,Y 199.689,Z 305.411,A -85,B 0,C 180,E1 -21388.135,E2 -21388.135} C_VEL
LIN {X 0,Y 199.681,Z 305.406,A -85,B 0,C 180,E1 -21392.771,E2 -21392.771} C_VEL
LIN {X 0,Y 199.708,Z 305.406,A -85,B 0,C 180,E1 -21397.226,E2 -21397.226} C_VEL
LIN {X 0,Y 199.79,Z 305.411,A -85,B 0,C 180,E1 -21401.758,E2 -21401.758} C_VEL
LIN {X 0,Y 199.828,Z 305.392,A -85,B 0,C 180,E1 -21405.748,E2 -21405.748} C_VEL
LIN {X 0,Y 200.017,Z 305.363,A -85,B 0,C 180,E1 -21409.882,E2 -21409.882} C_VEL
LIN {X 0,Y 200.018,Z 305.38,A -85,B 0,C 180,E1 -21413.949,E2 -21413.949} C_VEL
LIN {X 0,Y 200.312,Z 305.331,A -85,B 0,C 180,E1 -21417.99,E2 -21417.99} C_VEL
LIN {X 0,Y 200.472,Z 305.323,A -85,B 0,C 180,E1 -21420,E2 -21420} C_VEL
LIN {X 0,Y 200.01,Z 305.375,A -85,B 0,C 180,E1 -21424.03,E2 -21424.03} C_VEL
LIN {X 0,Y 200.068,Z 305.362,A -85,B 0,C 180,E1 -21428.078,E2 -21428.078} C_VEL
LIN {X 0,Y 199.867,Z 305.389,A -85,B 0,C 180,E1 -21432.18,E2 -21432.18} C_VEL
LIN {X 0,Y 199.797,Z 305.402,A -85,B 0,C 180,E1 -21436.344,E2 -21436.344} C_VEL
LIN {X 0,Y 199.695,Z 305.419,A -85,B 0,C 180,E1 -21440.606,E2 -21440.606} C_VEL
LIN {X 0,Y 199.746,Z 305.475,A -85,B 0,C 180,E1 -21443.541,E2 -21443.541} C_VEL
LIN {X 0,Y 200.65,Z 308.11,A -85,B 0,C 180,E1 -21443.955,E2 -21443.955} C_VEL
LIN {X 0,Y 202.923,Z 310.89,A -85,B 0,C 180,E1 -21444.762,E2 -21444.762} C_VEL
LIN {X 0,Y 205.302,Z 314.401,A -85,B 0,C 180,E1 -21445.607,E2 -21445.607} C_VEL
LIN {X 0,Y 211.021,Z 323.673,A -85,B 0,C 180,E1 -21447.523,E2 -21447.523} C_VEL
LIN {X 0,Y 216.039,Z 333.396,A -85,B 0,C 180,E1 -21449.147,E2 -21449.147} C_VEL
LIN {X 0,Y 220.86,Z 344.567,A -85,B 0,C 180,E1 -21450.66,E2 -21450.66} C_VEL
LIN {X 0,Y 221.191,Z 345.546,A -85,B 0,C 180,E1 -21450.769,E2 -21450.769} C_VEL
LIN {X 0,Y 219.294,Z 380.548,A -85,B 0,C 180,E1 -21451.987,E2 -21451.987} C_VEL
LIN {X 0,Y 218.356,Z 390.421,A -85,B 0,C 180,E1 -21452.556,E2 -21452.556} C_VEL
LIN {X 0,Y 216.89,Z 401.463,A -85,B 0,C 180,E1 -21453.516,E2 -21453.516} C_VEL
LIN {X 0,Y 214.906,Z 411.644,A -85,B 0,C 180,E1 -21454.763,E2 -21454.763} C_VEL
LIN {X 0,Y 212.907,Z 420.094,A -85,B 0,C 180,E1 -21456.108,E2 -21456.108} C_VEL
LIN {X 0,Y 210.852,Z 427.837,A -85,B 0,C 180,E1 -21457.665,E2 -21457.665} C_VEL
LIN {X 0,Y 208.818,Z 434.414,A -85,B 0,C 180,E1 -21459.28,E2 -21459.28} C_VEL
LIN {X 0,Y 206.877,Z 440.086,A -85,B 0,C 180,E1 -21460.967,E2 -21460.967} C_VEL
LIN {X 0,Y 204.715,Z 445.859,A -85,B 0,C 180,E1 -21463.079,E2 -21463.079} C_VEL
LIN {X 0,Y 202.803,Z 450.94,A -85,B 0,C 180,E1 -21465.434,E2 -21465.434} C_VEL
LIN {X 0,Y 200.833,Z 455.729,A -85,B 0,C 180,E1 -21468.328,E2 -21468.328} C_VEL
LIN {X 0,Y 199.513,Z 458.691,A -85,B 0,C 180,E1 -21470.802,E2 -21470.802} C_VEL
LIN {X 0,Y 198.541,Z 460.562,A -85,B 0,C 180,E1 -21473.005,E2 -21473.005} C_VEL
LIN {X 0,Y 197.863,Z 461.879,A -85,B 0,C 180,E1 -21475.369,E2 -21475.369} C_VEL
LIN {X 0,Y 197.171,Z 462.665,A -85,B 0,C 180,E1 -21478.811,E2 -21478.811} C_VEL
LIN {X 0,Y 196.933,Z 461.482,A -85,B 0,C 180,E1 -21483.149,E2 -21483.149} C_VEL
LIN {X 0,Y 197.045,Z 460.595,A -85,B 0,C 180,E1 -21484.66,E2 -21484.66} C_VEL
LIN {X 0,Y 197.557,Z 457.85,A -85,B 0,C 180,E1 -21487.66,E2 -21487.66} C_VEL
LIN {X 0,Y 198.105,Z 454.409,A -85,B 0,C 180,E1 -21490.305,E2 -21490.305} C_VEL
LIN {X 0,Y 198.828,Z 450.475,A -85,B 0,C 180,E1 -21492.626,E2 -21492.626} C_VEL
LIN {X 0,Y 199.866,Z 444.867,A -85,B 0,C 180,E1 -21495.231,E2 -21495.231} C_VEL
LIN {X 0,Y 201.338,Z 437.491,A -85,B 0,C 180,E1 -21497.911,E2 -21497.911} C_VEL
LIN {X 0,Y 202.925,Z 428.887,A -85,B 0,C 180,E1 -21500.28,E2 -21500.28} C_VEL
LIN {X 0,Y 204.154,Z 421.891,A -85,B 0,C 180,E1 -21501.837,E2 -21501.837} C_VEL
LIN {X 0,Y 205.476,Z 413.732,A -85,B 0,C 180,E1 -21503.308,E2 -21503.308} C_VEL
LIN {X 0,Y 206.513,Z 406.367,A -85,B 0,C 180,E1 -21504.385,E2 -21504.385} C_VEL
LIN {X 0,Y 207.416,Z 397.817,A -85,B 0,C 180,E1 -21505.384,E2 -21505.384} C_VEL
LIN {X 0,Y 208.281,Z 388.328,A -85,B 0,C 180,E1 -21506.203,E2 -21506.203} C_VEL
LIN {X 0,Y 208.921,Z 378.88,A -85,B 0,C 180,E1 -21506.753,E2 -21506.753} C_VEL
LIN {X 0,Y 210.333,Z 338.026,A -85,B 0,C 180,E1 -21508.235,E2 -21508.235} C_VEL
LIN {X 0,Y 208.806,Z 329.166,A -85,B 0,C 180,E1 -21508.741,E2 -21508.741} C_VEL
LIN {X 0,Y 202.794,Z 311.383,A -85,B 0,C 180,E1 -21510.13,E2 -21510.13} C_VEL
LIN {X 0,Y 200.505,Z 305.948,A -85,B 0,C 180,E1 -21510.628,E2 -21510.628} C_VEL
LIN {X 0,Y 200.394,Z 305.337,A -85,B 0,C 180,E1 -21510.754,E2 -21510.754} C_VEL
LIN {X 0,Y 200.017,Z 305.377,A -85,B 0,C 180,E1 -21516.051,E2 -21516.051} C_VEL
LIN {X 0,Y 200.024,Z 305.38,A -85,B 0,C 180,E1 -21520.118,E2 -21520.118} C_VEL
LIN {X 0,Y 199.825,Z 305.401,A -85,B 0,C 180,E1 -21524.252,E2 -21524.252} C_VEL
LIN {X 0,Y 199.78,Z 305.407,A -85,B 0,C 180,E1 -21528.457,E2 -21528.457} C_VEL
LIN {X 0,Y 199.715,Z 305.41,A -85,B 0,C 180,E1 -21533.802,E2 -21533.802} C_VEL
LIN {X 0,Y 199.713,Z 305.423,A -85,B 0,C 180,E1 -21538.386,E2 -21538.386} C_VEL
LIN {X 0,Y 199.677,Z 305.419,A -85,B 0,C 180,E1 -21542.357,E2 -21542.357} C_VEL
LIN {X 0,Y 199.622,Z 305.432,A -85,B 0,C 180,E1 -21546.762,E2 -21546.762} C_VEL
LIN {X 0,Y 199.608,Z 305.432,A -85,B 0,C 180,E1 -21549.327,E2 -21549.327} C_VEL
LIN {X 0,Y 199.619,Z 305.425,A -85,B 0,C 180,E1 -21554.758,E2 -21554.758} C_VEL
LIN {X 0,Y 199.654,Z 305.427,A -85,B 0,C 180,E1 -21558.024,E2 -21558.024} C_VEL
LIN {X 0,Y 199.677,Z 305.42,A -85,B 0,C 180,E1 -21560.742,E2 -21560.742} C_VEL
LIN {X 0,Y 199.631,Z 305.413,A -85,B 0,C 180,E1 -21565.717,E2 -21565.717} C_VEL
LIN {X 0,Y 199.7,Z 305.416,A -85,B 0,C 180,E1 -21568.137,E2 -21568.137} C_VEL
LIN {X 0,Y 199.683,Z 305.422,A -85,B 0,C 180,E1 -21572.771,E2 -21572.771} C_VEL
LIN {X 0,Y 199.733,Z 305.404,A -85,B 0,C 180,E1 -21577.228,E2 -21577.228} C_VEL
LIN {X 0,Y 199.792,Z 305.397,A -85,B 0,C 180,E1 -21581.757,E2 -21581.757} C_VEL
LIN {X 0,Y 199.829,Z 305.403,A -85,B 0,C 180,E1 -21585.748,E2 -21585.748} C_VEL
LIN {X 0,Y 200.018,Z 305.378,A -85,B 0,C 180,E1 -21589.881,E2 -21589.881} C_VEL
LIN {X 0,Y 200.015,Z 305.364,A -85,B 0,C 180,E1 -21593.949,E2 -21593.949} C_VEL
LIN {X 0,Y 200.313,Z 305.335,A -85,B 0,C 180,E1 -21597.989,E2 -21597.989} C_VEL
LIN {X 0,Y 200.472,Z 305.321,A -85,B 0,C 180,E1 -21600,E2 -21600} C_VEL
LIN {X 0,Y 200.018,Z 305.379,A -85,B 0,C 180,E1 -21604.029,E2 -21604.029} C_VEL
LIN {X 0,Y 200.082,Z 305.359,A -85,B 0,C 180,E1 -21608.077,E2 -21608.077} C_VEL
LIN {X 0,Y 199.868,Z 305.395,A -85,B 0,C 180,E1 -21612.18,E2 -21612.18} C_VEL
LIN {X 0,Y 199.797,Z 305.408,A -85,B 0,C 180,E1 -21616.344,E2 -21616.344} C_VEL
LIN {X 0,Y 199.676,Z 305.413,A -85,B 0,C 180,E1 -21620.608,E2 -21620.608} C_VEL
LIN {X 0,Y 199.659,Z 305.425,A -85,B 0,C 180,E1 -21624.986,E2 -21624.986} C_VEL
LIN {X 0,Y 199.66,Z 305.422,A -85,B 0,C 180,E1 -21629.524,E2 -21629.524} C_VEL
LIN {X 0,Y 199.667,Z 305.424,A -85,B 0,C 180,E1 -21632.356,E2 -21632.356} C_VEL
LIN {X 0,Y 199.619,Z 305.429,A -85,B 0,C 180,E1 -21636.764,E2 -21636.764} C_VEL
LIN {X 0,Y 199.604,Z 305.42,A -85,B 0,C 180,E1 -21639.329,E2 -21639.329} C_VEL
LIN {X 0,Y 199.571,Z 305.423,A -85,B 0,C 180,E1 -21642.311,E2 -21642.311} C_VEL
LIN {X 0,Y 199.578,Z 305.437,A -85,B 0,C 180,E1 -21645.23,E2 -21645.23} C_VEL
LIN {X 0,Y 199.577,Z 305.436,A -85,B 0,C 180,E1 -21648.006,E2 -21648.006} C_VEL
LIN {X 0,Y 199.608,Z 305.434,A -85,B 0,C 180,E1 -21650.768,E2 -21650.768} C_VEL
LIN {X 0,Y 199.634,Z 305.428,A -85,B 0,C 180,E1 -21655.719,E2 -21655.719} C_VEL
LIN {X 0,Y 199.733,Z 305.553,A -85,B 0,C 180,E1 -21656.957,E2 -21656.957} C_VEL
LIN {X 0,Y 201.37,Z 313.682,A -85,B 0,C 180,E1 -21661.4,E2 -21661.4} C_VEL
LIN {X 0,Y 205.722,Z 327.224,A -85,B 0,C 180,E1 -21662.452,E2 -21662.452} C_VEL
LIN {X 0,Y 208.645,Z 349.977,A -85,B 0,C 180,E1 -21663.663,E2 -21663.663} C_VEL
LIN {X 0,Y 208.543,Z 355.81,A -85,B 0,C 180,E1 -21663.879,E2 -21663.879} C_VEL
LIN {X 0,Y 207.304,Z 361.614,A -85,B 0,C 180,E1 -21663.98,E2 -21663.98} C_VEL
LIN {X 0,Y 203.729,Z 373.124,A -85,B 0,C 180,E1 -21664.069,E2 -21664.069} C_VEL
LIN {X 0,Y 202.536,Z 379.002,A -85,B 0,C 180,E1 -21664.182,E2 -21664.182} C_VEL
LIN {X 0,Y 202.374,Z 380.986,A -85,B 0,C 180,E1 -21664.245,E2 -21664.245} C_VEL
LIN {X 0,Y 201.644,Z 396.018,A -85,B 0,C 180,E1 -21664.943,E2 -21664.943} C_VEL
LIN {X 0,Y 200.434,Z 406.498,A -85,B 0,C 180,E1 -21665.774,E2 -21665.774} C_VEL
LIN {X 0,Y 199.434,Z 415.842,A -85,B 0,C 180,E1 -21666.845,E2 -21666.845} C_VEL
LIN {X 0,Y 198.111,Z 424.573,A -85,B 0,C 180,E1 -21668.132,E2 -21668.132} C_VEL
LIN {X 0,Y 196.522,Z 433.791,A -85,B 0,C 180,E1 -21669.867,E2 -21669.867} C_VEL
LIN {X 0,Y 194.787,Z 443.054,A -85,B 0,C 180,E1 -21672.141,E2 -21672.141} C_VEL
LIN {X 0,Y 193.423,Z 449.645,A -85,B 0,C 180,E1 -21674.187,E2 -21674.187} C_VEL
LIN {X 0,Y 192.366,Z 455.127,A -85,B 0,C 180,E1 -21676.263,E2 -21676.263} C_VEL
LIN {X 0,Y 191.496,Z 459.694,A -85,B 0,C 180,E1 -21678.355,E2 -21678.355} C_VEL
LIN {X 0,Y 190.912,Z 463.491,A -85,B 0,C 180,E1 -21680.465,E2 -21680.465} C_VEL
LIN {X 0,Y 190.358,Z 467.79,A -85,B 0,C 180,E1 -21683.641,E2 -21683.641} C_VEL
LIN {X 0,Y 190.182,Z 470.276,A -85,B 0,C 180,E1 -21686.16,E2 -21686.16} C_VEL
LIN {X 0,Y 190.186,Z 471.578,A -85,B 0,C 180,E1 -21687.882,E2 -21687.882} C_VEL
LIN {X 0,Y 190.296,Z 472.574,A -85,B 0,C 180,E1 -21690,E2 -21690} C_VEL
LIN {X 0,Y 190.156,Z 473.187,A -85,B 0,C 180,E1 -21693.72,E2 -21693.72} C_VEL
LIN {X 0,Y 190.359,Z 472.671,A -85,B 0,C 180,E1 -21696.359,E2 -21696.359} C_VEL
LIN {X 0,Y 190.713,Z 471.668,A -85,B 0,C 180,E1 -21698.476,E2 -21698.476} C_VEL
LIN {X 0,Y 191.728,Z 469.255,A -85,B 0,C 180,E1 -21701.631,E2 -21701.631} C_VEL
LIN {X 0,Y 193.232,Z 465.525,A -85,B 0,C 180,E1 -21704.749,E2 -21704.749} C_VEL
LIN {X 0,Y 194.554,Z 462.364,A -85,B 0,C 180,E1 -21706.797,E2 -21706.797} C_VEL
LIN {X 0,Y 196.639,Z 457.35,A -85,B 0,C 180,E1 -21709.305,E2 -21709.305} C_VEL
LIN {X 0,Y 199.034,Z 451.077,A -85,B 0,C 180,E1 -21711.762,E2 -21711.762} C_VEL
LIN {X 0,Y 201.305,Z 444.957,A -85,B 0,C 180,E1 -21713.671,E2 -21713.671} C_VEL
